// TwinCAT 3 PLC project TwinCAT_OpenFramework_Core
// Title: TwinCAT Open Framework Core
// Company: Oleksandr Tiutyk FOP
// Author: Oleksandr Tiutyk
// ProjectVersion: 0.0.0.1
// Description: Core types and implementations for TwinCAT Open Framework: abstractions, enums, primitives, interfaces, base object, exceptions, collettions, etc.
// ProgramVersion: 3.1.4026.16
// libraries:
//   Tc2_Standard, * (Beckhoff Automation GmbH)
//   Tc2_System, * (Beckhoff Automation GmbH)
//   Tc2_Utilities, * (Beckhoff Automation GmbH)
//   Tc3_EventLogger, * (Beckhoff Automation GmbH)
//   Tc3_JsonXml, * (Beckhoff Automation GmbH)
//   Tc3_Module, * (Beckhoff Automation GmbH)
// project tree:
//   Abstractions/Interfaces/Action/ IAbortableAction.TcIO, IAction.TcIO
//   Abstractions/Interfaces/ ICloneable.TcIO, IDisposable.TcIO, IObject.TcIO
//   Abstractions/Interfaces/Process/ IAbortableProcess.TcIO, IProcess.TcIO
//   Abstractions/ Object.TcPOU
//   Collections/PointerBased/PointerDictionary/ IReadOnlyPointerDictionary.TcIO, PointerDictionary.TcPOU, PointerDictionaryEnumerator.TcPOU
//   Collections/ Enumerator.TcPOU, ICollection.TcIO, IEnumerable.TcIO, IEnumerator.TcIO, KEY_VALUE_POINTER_PAIR.TcDUT
//   Collections/PointerBased/PointerUniqueSet/ IReadOnlyPointerUniqueSet.TcIO, PointerUniqueSet.TcPOU, PointerUniqueSetEnumerator.TcPOU
//   Collections/PointerBased/PointerList/ IReadOnlyPointerList.TcIO, PointerList.TcPOU, PointerListEnumerator.TcPOU
//   Collections/ValueBased/ByteList/ ByteList.TcPOU, ByteListEnumerator.TcPOU, IByteList.TcIO, IReadOnlyByteList.TcIO
//   Comparing/ COMPARISION_RESULT.TcDUT, IComparable.TcIO, IComparer.TcIO, StandardComparers.TcPOU
//   Comparing/StandardComparers/ BoolComparer.TcPOU, ByteComparer.TcPOU, DateAndTimeComparer.TcPOU, UXIntComparer.TcPOU, XIntComparer.TcPOU, XWordComparer.TcPOU, LDateAndTimeComparer.TcPOU, DateComparer.TcPOU, DIntComparer.TcPOU, DWordComparer.TcPOU, IntComparer.TcPOU, LIntComparer.TcPOU, LRealComparer.TcPOU, LTimeComparer.TcPOU, LWordComparer.TcPOU, PointerComparer.TcPOU, RealComparer.TcPOU, SIntComparer.TcPOU, StringComparer.TcPOU, TimeComparer.TcPOU, TimeOfDayComparer.TcPOU, LTimeOfDayComparer.TcPOU, UDIntComparer.TcPOU, UIntComparer.TcPOU, ULIntComparer.TcPOU, USIntComparer.TcPOU, WordComparer.TcPOU, WStringComparer.TcPOU
//   Enums/ EXECUTION_STATE.TcDUT, LOAD_STATE.TcDUT, POINTER_TYPE.TcDUT, SORTING_DIRECTION.TcDUT, TASK_STATE.TcDUT
//   Exceptions/Aggregate/ AggregateException.TcPOU
//   Exceptions/Empty/ EmptyException.TcPOU
//   Exceptions/ Exception.TcPOU, ExceptionManager.TcPOU, IException.TcIO
//   Exceptions/General/ArgumentOutOfRange/ ArgumentOutOfRangeException.TcPOU
//   Exceptions/General/ GeneralException.TcPOU
//   Exceptions/General/NotImplemented/ NotImplementedException.TcPOU
//   Exceptions/General/Standard/ StandardException.TcPOU
//   Exceptions/System/ SystemException.TcPOU
//   Helpers/ MathHelper.TcPOU
//   / CurrentNamespace.TcGVL
//   Internals/Statistics/ ObjectStatistics.TcPOU, ObjectStatisticsSettings.TcGVL, OBJECT_STATISTICS.TcDUT
//   Primitives/AnyType/ AnyTypeHelper.TcPOU
//   Primitives/Bit/ BitHelper.TcPOU
//   Primitives/Byte/ ByteHelper.TcPOU
//   Primitives/DateAndTime/ SystemDateTimeManager.TcPOU
//   Primitives/Pointer/ PointerHelper.TcPOU
//   Primitives/String/ StringBuilder.TcPOU, StringHelper.TcPOU
//   Primitives/WideString/ WideStringBuilder.TcPOU, WideStringHelper.TcPOU
//   Timers/ Timer.TcPOU
//   TypeAliases/ ERROR_MESSAGE.TcDUT, JSON_DOCUMENT.TcDUT

// ---- Collections/KEY_VALUE_POINTER_PAIR.TcDUT
TYPE KEY_VALUE_POINTER_PAIR :
STRUCT
	Key : PVOID;
	Value : PVOID;
END_STRUCT
END_TYPE

// ---- Comparing/COMPARISION_RESULT.TcDUT
{attribute 'qualified_only'}
{attribute 'strict'}
{attribute 'to_string'}
TYPE COMPARISION_RESULT :
(
	LEFT_LESS_RIGHT := -1,
	EQUALS := 0,
	LEFT_GREATER_RIGHT := 1
) SINT;
END_TYPE

// ---- Enums/EXECUTION_STATE.TcDUT
{attribute 'qualified_only'}
{attribute 'strict'}
{attribute 'to_string'}
// error should be reported using exceptions
TYPE EXECUTION_STATE :
(
	BUSY,
	DONE
);
END_TYPE

// ---- Enums/LOAD_STATE.TcDUT
{attribute 'qualified_only'}
{attribute 'strict'}
{attribute 'to_string'}
TYPE LOAD_STATE :
(
	NOT_LOADED,
	LOADING,
	LOADED,
	FAILED
);
END_TYPE

// ---- Enums/POINTER_TYPE.TcDUT
{attribute 'qualified_only'}
{attribute 'strict'}
{attribute 'to_string'}
TYPE POINTER_TYPE :
(
	BOOL_POINTER := 1,
	BYTE_POINTER := 2,
	WORD_POINTER := 3,
	DWORD_POINTER := 4,
	LWORD_POINTER := 5,
	SINT_POINTER := 6,
	USINT_POINTER := 7,
	INT_POINTER := 8,
	UINT_POINTER := 9,
	DINT_POINTER := 10,
	UDINT_POINTER := 11,
	LINT_POINTER := 12,
	ULINT_POINTER := 13,	
	XINT_POINTER := 14, 
	XWORD_POINTER := 15,	
	UXINT_POINTER := 16, 
	REAL_POINTER := 17,
	LREAL_POINTER := 18,
	STRING_POINTER := 19,
	WSTRING_POINTER := 20,
	TIME_POINTER := 21,
	LTIME_POINTER := 22,
	DATE_POINTER := 23,
	DATE_AND_TIME_POINTER := 24,
	LDATE_AND_TIME_POINTER := 25,
	TIME_OF_DAY_POINTER := 26,
	LTIME_OF_DAY_POINTER := 27,
	UNTYPED_POINTER := 28,
	OBJECT_POINTER := 29
) BYTE;
END_TYPE

// ---- Enums/SORTING_DIRECTION.TcDUT
{attribute 'qualified_only'}
{attribute 'strict'}
{attribute 'to_string'}
TYPE SORTING_DIRECTION :
(
	ASCENDING,
	DESCENDING
);
END_TYPE

// ---- Enums/TASK_STATE.TcDUT
{attribute 'qualified_only'}
{attribute 'strict'}
{attribute 'to_string'}
TYPE TASK_STATE :
(
	IDLE,
	EXECUTING,	
	DONE,
	ERROR,
	ABORTING,
	ABORTED
);
END_TYPE

// ---- Internals/Statistics/OBJECT_STATISTICS.TcDUT
TYPE OBJECT_STATISTICS :
STRUCT
	TypeName : STRING(255);
	InstanceCount : LINT;
END_STRUCT
END_TYPE

// ---- TypeAliases/ERROR_MESSAGE.TcDUT
TYPE ERROR_MESSAGE : WSTRING(2000); END_TYPE

// ---- TypeAliases/JSON_DOCUMENT.TcDUT
TYPE JSON_DOCUMENT : STRING(25000); END_TYPE

// ---- CurrentNamespace.TcGVL
{attribute 'qualified_only'}
VAR_GLOBAL
	{attribute 'OPC.UA.DA' := '1'}
	{attribute 'OPC.UA.DA.Access' := '1'}
	{attribute 'init_namespace'} 
	Name : STRING(255);	
END_VAR

// ---- Internals/Statistics/ObjectStatisticsSettings.TcGVL
{attribute 'qualified_only'}
VAR_GLOBAL PERSISTENT
	{attribute 'OPC.UA.DA' := '1'}	
	// Indicates if object creating and deleting counted in ObjectStatistics
	CountObjectStatistics : BOOL;
END_VAR

// ---- Abstractions/Interfaces/Action/IAbortableAction.TcIO
INTERFACE IAbortableAction EXTENDS IAction

{attribute 'monitoring' := 'call'}
{attribute 'OPC.UA.DA.Property' := '1'}
{attribute 'OPC.UA.DA.Access' := '1'}
PROPERTY Aborted : BOOL
GET
END_GET
END_PROPERTY

{attribute 'monitoring' := 'call'}
{attribute 'OPC.UA.DA.Property' := '1'}
{attribute 'OPC.UA.DA.Access' := '1'}
PROPERTY Aborting : BOOL
GET
END_GET
END_PROPERTY

{attribute 'monitoring' := 'call'}
{attribute 'OPC.UA.DA.Property' := '1'}
{attribute 'OPC.UA.DA.Access' := '1'}
PROPERTY AbortReason : REFERENCE TO ERROR_MESSAGE
GET
END_GET
END_PROPERTY

METHOD RequestAbort
VAR_INPUT 
	reason : ERROR_MESSAGE;
END_VAR
END_METHOD

END_INTERFACE

// ---- Abstractions/Interfaces/Action/IAction.TcIO
INTERFACE IAction EXTENDS IObject

{attribute 'monitoring' := 'call'}
{attribute 'OPC.UA.DA.Property' := '1'}
{attribute 'OPC.UA.DA.Access' := '1'}
PROPERTY Busy : BOOL
GET
END_GET
END_PROPERTY

{attribute 'monitoring' := 'call'}
{attribute 'OPC.UA.DA.Property' := '1'}
{attribute 'OPC.UA.DA.Access' := '1'}
PROPERTY Done : BOOL
GET
END_GET
END_PROPERTY

{attribute 'monitoring' := 'call'}
{attribute 'OPC.UA.DA.Property' := '1'}
{attribute 'OPC.UA.DA.Access' := '1'}
PROPERTY Error : BOOL
GET
END_GET
END_PROPERTY

METHOD Execute
END_METHOD

END_INTERFACE

// ---- Abstractions/Interfaces/ICloneable.TcIO
INTERFACE ICloneable EXTENDS __System.IQueryInterface

METHOD Clone : IObject
END_METHOD

END_INTERFACE

// ---- Abstractions/Interfaces/IDisposable.TcIO
INTERFACE IDisposable EXTENDS __System.IQueryInterface

METHOD Dispose
END_METHOD

END_INTERFACE

// ---- Abstractions/Interfaces/IObject.TcIO
INTERFACE IObject EXTENDS __System.IQueryInterface, IDisposable

{attribute 'monitoring' := 'call'}
PROPERTY ClassName : STRING
GET
END_GET
END_PROPERTY

{attribute "object_name" := "Equals"}
METHOD Equals : BOOL
VAR_INPUT 
	object : IObject;
END_VAR
END_METHOD

END_INTERFACE

// ---- Abstractions/Interfaces/Process/IAbortableProcess.TcIO
INTERFACE IAbortableProcess EXTENDS IProcess

{attribute 'monitoring' := 'call'}
{attribute 'OPC.UA.DA.Property' := '1'}
{attribute 'OPC.UA.DA.Access' := '1'}
PROPERTY Aborted : BOOL
GET
END_GET
END_PROPERTY

{attribute 'monitoring' := 'call'}
{attribute 'OPC.UA.DA.Property' := '1'}
{attribute 'OPC.UA.DA.Access' := '1'}
PROPERTY AbortReason : REFERENCE TO ERROR_MESSAGE
GET
END_GET
END_PROPERTY

{attribute 'monitoring' := 'call'}
{attribute 'OPC.UA.DA.Property' := '1'}
{attribute 'OPC.UA.DA.Access' := '1'}
PROPERTY Busy : BOOL
GET
END_GET
END_PROPERTY

METHOD RequestAbort
VAR_INPUT 
	reason : ERROR_MESSAGE;
END_VAR
END_METHOD

END_INTERFACE

// ---- Abstractions/Interfaces/Process/IProcess.TcIO
INTERFACE IProcess EXTENDS IObject

{attribute 'monitoring' := 'call'}
{attribute 'OPC.UA.DA.Property' := '1'}
{attribute 'OPC.UA.DA.Access' := '1'}
PROPERTY Busy : BOOL
GET
END_GET
END_PROPERTY

{attribute 'monitoring' := 'call'}
{attribute 'OPC.UA.DA.Property' := '1'}
{attribute 'OPC.UA.DA.Access' := '1'}
PROPERTY Error : BOOL
GET
END_GET
END_PROPERTY

METHOD Execute
END_METHOD

END_INTERFACE

// ---- Collections/PointerBased/PointerDictionary/IReadOnlyPointerDictionary.TcIO
INTERFACE IReadOnlyPointerDictionary EXTENDS ICollection

METHOD ContainsKey : BOOL
VAR_INPUT
	key : PVOID;
END_VAR
END_METHOD

METHOD GetKeyByIndex : PVOID
VAR_INPUT
	index : DINT;
END_VAR
END_METHOD

METHOD GetValueByIndex : PVOID
VAR_INPUT
	index : DINT;
END_VAR
END_METHOD

METHOD GetValueByKey : PVOID
VAR_INPUT
	key : PVOID;
END_VAR
END_METHOD

{attribute 'OPC.UA.DA.Property' := '1'}
{attribute 'monitoring' := 'call'}
PROPERTY KeyType : POINTER_TYPE
GET
END_GET
END_PROPERTY

{attribute 'OPC.UA.DA.Property' := '1'}
{attribute 'monitoring' := 'call'}
PROPERTY ValueType : POINTER_TYPE
GET
END_GET
END_PROPERTY

END_INTERFACE

// ---- Collections/PointerBased/PointerUniqueSet/IReadOnlyPointerUniqueSet.TcIO
INTERFACE IReadOnlyPointerUniqueSet EXTENDS ICollection

METHOD Contains : BOOL
VAR_INPUT
	element : PVOID;
END_VAR
END_METHOD

{attribute 'OPC.UA.DA.Property' := '1'}
{attribute 'monitoring' := 'call'}
PROPERTY ElementType : POINTER_TYPE
GET
END_GET
END_PROPERTY

METHOD GetByIndex : PVOID
VAR_INPUT
	index : DINT;
END_VAR
END_METHOD

END_INTERFACE

// ---- Collections/ICollection.TcIO
INTERFACE ICollection EXTENDS IEnumerable

{attribute 'OPC.UA.DA.Property' := '1'}
{attribute 'monitoring' := 'call'}
PROPERTY Count : DINT
GET
END_GET
END_PROPERTY

END_INTERFACE

// ---- Collections/IEnumerable.TcIO
INTERFACE IEnumerable EXTENDS IObject

METHOD GetDefaultEnumerator : IEnumerator
END_METHOD

END_INTERFACE

// ---- Collections/IEnumerator.TcIO
INTERFACE IEnumerator EXTENDS IObject

// Shows curent collection element
PROPERTY ABSTRACT Current : PVOID
GET
END_GET
END_PROPERTY

// Moves Current pointer to next collection element
METHOD MoveNext : BOOL
END_METHOD

// Sets the enumerator to its initial position, which is before the first element in the collection
METHOD Reset
END_METHOD

END_INTERFACE

// ---- Collections/PointerBased/PointerList/IReadOnlyPointerList.TcIO
INTERFACE IReadOnlyPointerList EXTENDS ICollection

{attribute 'OPC.UA.DA.Property' := '1'}
{attribute 'monitoring' := 'call'}
PROPERTY ElementType : POINTER_TYPE
GET
END_GET
END_PROPERTY

METHOD Find : BOOL
VAR_INPUT
	pattern : PVOID;
	comparer : IComparer;
	skip : DINT;
END_VAR
VAR_OUTPUT
	element : PVOID;
	index : DINT;
END_VAR
END_METHOD

METHOD Get : PVOID
VAR_INPUT
	index : DINT;
END_VAR
END_METHOD

METHOD Sort
VAR_INPUT
	comparer : IComparer;
	direction : SORTING_DIRECTION;
END_VAR
END_METHOD

END_INTERFACE

// ---- Collections/ValueBased/ByteList/IByteList.TcIO
INTERFACE IByteList EXTENDS IReadOnlyByteList

METHOD Set
VAR_INPUT
	index : DINT;
	value : BYTE;
END_VAR
END_METHOD

END_INTERFACE

// ---- Collections/ValueBased/ByteList/IReadOnlyByteList.TcIO
INTERFACE IReadOnlyByteList EXTENDS ICollection

{attribute 'OPC.UA.DA.Property' := '1'}
{attribute 'monitoring' := 'call'}
PROPERTY Address : POINTER TO BYTE
GET
END_GET
END_PROPERTY

METHOD Get : BYTE
VAR_INPUT
	index : DINT;
END_VAR
END_METHOD

END_INTERFACE

// ---- Comparing/IComparable.TcIO
INTERFACE IComparable EXTENDS IObject

METHOD CompareTo : COMPARISION_RESULT
VAR_INPUT
	object : IObject;
END_VAR
END_METHOD

END_INTERFACE

// ---- Comparing/IComparer.TcIO
INTERFACE IComparer EXTENDS IObject

METHOD Compare : COMPARISION_RESULT
VAR_INPUT
	left : PVOID;
	right : PVOID;
END_VAR
END_METHOD

END_INTERFACE

// ---- Exceptions/IException.TcIO
INTERFACE IException EXTENDS ICloneable, IDisposable

{attribute 'monitoring' := 'call'}
PROPERTY Empty : BOOL
GET
END_GET
END_PROPERTY

// Work is not possible after such error
{attribute 'monitoring' := 'call'}
PROPERTY Fatal : BOOL
GET
END_GET
END_PROPERTY

METHOD ABSTRACT GetMessage : ERROR_MESSAGE
VAR_INPUT
	showTimestamp : BOOL := FALSE;
	showSource : BOOL := FALSE;
END_VAR
END_METHOD

METHOD GetSourceDescription : WSTRING(300)
END_METHOD

{attribute 'monitoring' := 'call'}
PROPERTY LocalTimestamp : DATE_AND_TIME
GET
END_GET
END_PROPERTY

{attribute 'monitoring' := 'call'}
PROPERTY SourceClassName : STRING
GET
END_GET
END_PROPERTY

{attribute 'monitoring' := 'call'}
PROPERTY SourceMethodName : STRING
GET
END_GET
END_PROPERTY

{attribute 'monitoring' := 'call'}
PROPERTY SourceNamespaceName : STRING
GET
END_GET
END_PROPERTY

{attribute 'monitoring' := 'call'}
PROPERTY SourcePosition : STRING
GET
END_GET
END_PROPERTY

{attribute 'monitoring' := 'call'}
PROPERTY UtcTimestamp : DATE_AND_TIME
GET
END_GET
END_PROPERTY

END_INTERFACE

// ---- Abstractions/Object.TcPOU
{attribute 'no_explicit_call' := 'Direct call is not allowed'} 
FUNCTION_BLOCK ABSTRACT Object IMPLEMENTS IObject

{attribute 'monitoring' := 'call'}
PROPERTY ABSTRACT ClassName : STRING
GET
END_GET
END_PROPERTY

METHOD Dispose
VAR
	self : POINTER TO Object;
END_VAR
PointerHelper.ReleaseDynamicMemory(THIS, POINTER_TYPE.OBJECT_POINTER);
END_METHOD

{attribute "object_name" := "Equals"}
METHOD Equals : BOOL
VAR_INPUT 
	object : IObject;
END_VAR
VAR
	selfPointer : POINTER TO Object;
	comparingPointer : POINTER TO Object;
END_VAR
selfPointer := THIS;

IF __QUERYPOINTER(object, comparingPointer) THEN
	Equals := selfPointer = comparingPointer;
END_IF
END_METHOD

METHOD FB_exit : BOOL
VAR_INPUT
	bInCopyCode : BOOL; // if TRUE, the exit method is called for exiting an instance that is copied afterwards (online change).
END_VAR
IF ObjectStatisticsSettings.CountObjectStatistics THEN
	ObjectStatistics.RemoveObject(THIS^);
END_IF
END_METHOD

METHOD FB_init : BOOL
VAR_INPUT
	bInitRetains : BOOL; // if TRUE, the retain variables are initialized (warm start / cold start)
	bInCopyCode : BOOL; // if TRUE, the instance afterwards gets moved into the copy code (online change)
END_VAR
IF ObjectStatisticsSettings.CountObjectStatistics THEN
	ObjectStatistics.AddObject(THIS^);
END_IF
END_METHOD

END_FUNCTION_BLOCK

// ---- Primitives/Pointer/PointerHelper.TcPOU
PROGRAM PointerHelper

METHOD ReleaseDynamicMemory
VAR_INPUT
	value : POINTER TO BYTE;
	pointerType : POINTER_TYPE;
END_VAR
VAR
	memoryArea : Tc2_System.E_TcMemoryArea;
	objectPointer : POINTER TO Object;
END_VAR
IF value = 0 THEN
	RETURN;
END_IF

// check at list first byte of released memory
memoryArea := Tc2_System.F_CheckMemoryArea(value, 1);

IF memoryArea <> E_TcMemoryArea.Dynamic THEN
	RETURN;
END_IF

IF pointerType = POINTER_TYPE.OBJECT_POINTER THEN
	objectPointer := value;
	// to call FB_exit
	__DELETE(objectPointer);
ELSE
	__DELETE(value);
END_IF
END_METHOD

END_PROGRAM

// ---- Internals/Statistics/ObjectStatistics.TcPOU
{attribute 'no_explicit_call' := 'Direct call is not allowed'} 
PROGRAM ObjectStatistics
VAR CONSTANT
	{attribute 'OPC.UA.DA' := '1'}
	{attribute 'OPC.UA.DA.Access' := '1'}	
	OBJECT_STATISTICS_BUFFER_SIZE : DINT := 1000;
END_VAR
VAR_OUTPUT
	{attribute 'OPC.UA.DA' := '1'}
	{attribute 'OPC.UA.DA.Access' := '1'}	
	CreateObjectCounter : DWORD; // Increments each time when object created
	{attribute 'OPC.UA.DA' := '1'}
	{attribute 'OPC.UA.DA.Access' := '1'}	
	DeleteObjectCounter : DWORD; // Decrements each time when object created
	{attribute 'OPC.UA.DA' := '1'}
	{attribute 'OPC.UA.DA.Access' := '1'}	
	ObjectCount : LINT; // Count of existing objecs
	{attribute 'OPC.UA.DA' := '1'}
	{attribute 'OPC.UA.DA.Access' := '1'}	
	ObjectStatistics : ARRAY [0..OBJECT_STATISTICS_BUFFER_SIZE - 1] OF OBJECT_STATISTICS;
END_VAR

METHOD INTERNAL AddObject : BOOL
VAR_IN_OUT CONSTANT
	object : Object;
END_VAR
VAR
	i : DINT;
END_VAR
IF CreateObjectCounter < 4294967295 THEN
	CreateObjectCounter := CreateObjectCounter + 1;
ELSE
	CreateObjectCounter := 0;
END_IF

ObjectCount := ObjectCount + 1;

IF object.ClassName = '' THEN
	RETURN;	
END_IF

FOR i := 0 TO OBJECT_STATISTICS_BUFFER_SIZE - 1 DO
	IF ObjectStatistics[i].TypeName = object.ClassName THEN		
		ObjectStatistics[i].InstanceCount := ObjectStatistics[i].InstanceCount + 1;		
		RETURN;
	ELSIF ObjectStatistics[i].TypeName = '' THEN	
		ObjectStatistics[i].TypeName := object.ClassName;
		ObjectStatistics[i].InstanceCount := 1;		
		RETURN;
	END_IF
END_FOR
END_METHOD

METHOD INTERNAL RemoveObject
VAR_IN_OUT CONSTANT
	object : Object;
END_VAR
VAR
	i : DINT;
END_VAR
IF DeleteObjectCounter < 4294967295 THEN
	DeleteObjectCounter := DeleteObjectCounter + 1;
ELSE
	DeleteObjectCounter := 0;
END_IF

ObjectCount := ObjectCount - 1;

IF object.ClassName = '' THEN
	RETURN;	
END_IF

FOR i := 0 TO OBJECT_STATISTICS_BUFFER_SIZE - 1 DO
	IF ObjectStatistics[i].TypeName = object.ClassName THEN				
		ObjectStatistics[i].InstanceCount := ObjectStatistics[i].InstanceCount - 1;
						
		RETURN;
	END_IF 
END_FOR
END_METHOD

END_PROGRAM

// ---- Collections/PointerBased/PointerDictionary/PointerDictionary.TcPOU
{attribute 'no_explicit_call' := 'do not call this function block directly'} 
// Dynamic dictionary of pointers to key and value
FUNCTION_BLOCK PointerDictionary EXTENDS Object IMPLEMENTS IReadOnlyPointerDictionary
VAR
	_ClassName : STRING := __POUNAME();
	_Keys : POINTER TO PVOID;
	_Values : POINTER TO PVOID;
	_ArrayLength : DINT;
	_ElementCount : DINT;
	_DefaultAllocationElemetsCount : BYTE := 10;
	_KeyType : POINTER_TYPE := POINTER_TYPE.BYTE_POINTER;
	_ValueType : POINTER_TYPE := POINTER_TYPE.BYTE_POINTER;
	_KeyComparer : IComparer;
	_DefaultEnumerator : PointerDictionaryEnumerator;
END_VAR

METHOD AllocateMemory
VAR_INPUT
	elementsCount : DINT;
END_VAR
VAR
	newKeys : POINTER TO PVOID;
	newValues : POINTER TO PVOID;
END_VAR
newKeys := __NEW(PVOID, TO_UDINT(_ArrayLength + elementsCount));
newValues := __NEW(PVOID, TO_UDINT(_ArrayLength + elementsCount));

IF _ElementCount > 0 THEN
	Tc2_System.MEMCPY(newKeys, _Keys, SIZEOF(POINTER TO BYTE) * TO_UDINT(_ElementCount)); 
	Tc2_System.MEMCPY(newValues, _Values, SIZEOF(POINTER TO BYTE) * TO_UDINT(_ElementCount));
END_IF

IF _Keys <> 0 THEN
	__DELETE(_Keys);
END_IF

IF _Values <> 0 THEN
	__DELETE(_Values);
END_IF
 
_Keys := newKeys;
_Values := newValues;
 
_ArrayLength := _ArrayLength + elementsCount;
END_METHOD

{attribute 'monitoring' := 'call'}
PROPERTY ClassName : STRING
GET
ClassName := _ClassName;
END_GET
END_PROPERTY

METHOD Clear
VAR_INPUT
	deleteKeys : BOOL;
	deleteValues : BOOL;
END_VAR
VAR
	i : DINT;
	value : PVOID;
END_VAR
IF deleteKeys AND_THEN _ElementCount > 0 THEN
	FOR i := 0 TO _ElementCount - 1 DO
		PointerHelper.ReleaseDynamicMemory(_Keys[i], _KeyType);						
	END_FOR	
END_IF

IF deleteValues AND_THEN _ElementCount > 0 THEN
	FOR i := 0 TO _ElementCount - 1 DO
		PointerHelper.ReleaseDynamicMemory(_Values[i], _ValueType);							
	END_FOR	
END_IF

IF _Keys <> 0 THEN
	__DELETE(_Keys);
END_IF

IF _Values <> 0 THEN
	__DELETE(_Values);
END_IF

_ElementCount := 0;
_ArrayLength := 0;
END_METHOD

METHOD ContainsKey : BOOL
VAR_INPUT
	key : PVOID;
END_VAR
VAR
	index : DINT; 
END_VAR
ContainsKey := SearchKeyPosition(key, supposedIndex => index);
END_METHOD

{attribute 'OPC.UA.DA.Property' := '1'}
{attribute 'monitoring' := 'call'}
PROPERTY Count : DINT
GET
Count := _ElementCount;
END_GET
END_PROPERTY

METHOD FB_exit : BOOL
VAR_INPUT
	bInCopyCode : BOOL; // if TRUE, the exit method is called for exiting an instance that is copied afterwards (online change).
END_VAR
Clear(FALSE, FALSE);
END_METHOD

METHOD FB_init : BOOL
VAR_INPUT
	bInitRetains : BOOL; // if TRUE, the retain variables are initialized (warm start / cold start)
	bInCopyCode : BOOL; // if TRUE, the instance afterwards gets moved into the copy code (online change)
	keyType : POINTER_TYPE;
	valueType : POINTER_TYPE;
	keyComparer : IComparer;
END_VAR
_DefaultEnumerator.Initialize(THIS^);

_KeyType := keyType;
_ValueType := valueType;

IF keyComparer = 0 THEN
	_KeyComparer := StandardComparers.GetForType(keyType);
ELSE
	_KeyComparer := keyComparer;
END_IF
END_METHOD

METHOD GetDefaultEnumerator : IEnumerator
GetDefaultEnumerator := _DefaultEnumerator;
END_METHOD

METHOD GetKeyByIndex : PVOID
VAR_INPUT
	index : DINT;
END_VAR
IF index >= 0 AND index < _ElementCount THEN
	GetKeyByIndex := _Keys[index];
END_IF
END_METHOD

METHOD GetValueByIndex : PVOID
VAR_INPUT
	index : DINT;
END_VAR
IF index >= 0 AND index < _ElementCount THEN
	GetValueByIndex := _Values[index];
END_IF
END_METHOD

METHOD GetValueByKey : PVOID
VAR_INPUT
	key : PVOID;
END_VAR
VAR
	index : DINT; 
END_VAR
IF SearchKeyPosition(key, supposedIndex => index) THEN
	GetValueByKey := _Values[index];
END_IF
END_METHOD

{attribute 'OPC.UA.DA.Property' := '1'}
{attribute 'monitoring' := 'call'}
PROPERTY KeyType : POINTER_TYPE
GET
KeyType := _KeyType;
END_GET
END_PROPERTY

METHOD Remove : BOOL
VAR_INPUT
	key : PVOID;
	deleteKey : BOOL;
	deleteValue : BOOL;
END_VAR
VAR
	index : DINT;
END_VAR
IF SearchKeyPosition(key, supposedIndex => index) THEN
	RemoveAt(index, deleteKey, deleteValue);
	Remove := TRUE;
END_IF
END_METHOD

METHOD RemoveAt : BOOL
VAR_INPUT
	index : DINT;
	deleteKey : BOOL;
	deleteValue : BOOL;
END_VAR
VAR
	i : DINT;
END_VAR
IF index < _ElementCount THEN
	IF deleteKey THEN
		PointerHelper.ReleaseDynamicMemory(_Keys[index], _KeyType);			
	END_IF
	
	IF deleteValue THEN
		PointerHelper.ReleaseDynamicMemory(_Values[index], _ValueType);			
	END_IF
	
	IF index + 2 <= _ElementCount THEN
		FOR	i := index TO _ElementCount - 2 DO
			_Keys[i] := _Keys[i + 1];
			_Values[i] := _Values[i + 1];
		END_FOR			
	END_IF
		
	_Keys[_ElementCount - 1] := 0;
	_Values[_ElementCount - 1] := 0;
	_ElementCount := _ElementCount - 1;
	
	RemoveAt := TRUE;
END_IF
END_METHOD

METHOD PROTECTED SearchKeyPosition : BOOL
VAR_INPUT
	key : PVOID;
END_VAR
VAR_OUTPUT
	supposedIndex : DINT; 
END_VAR
VAR
	lastIndex : DINT;
	minIndex : DINT;
	maxIndex : DINT;
END_VAR
IF _ElementCount = 0 THEN
	RETURN;
END_IF

lastIndex := _ElementCount - 1;
maxIndex := lastIndex;
supposedIndex := maxIndex / 2;

WHILE minIndex <= maxIndex DO
	CASE _KeyComparer.Compare(_Keys[supposedIndex], key) OF
		// assumed key equals to seached 
		COMPARISION_RESULT.EQUALS:
			SearchKeyPosition := TRUE;
			RETURN;

		// assumed key less than searched, move range to right
		COMPARISION_RESULT.LEFT_LESS_RIGHT:
			minIndex := supposedIndex + 1;
			
		// assumed key greater than searched, move range to left	
		COMPARISION_RESULT.LEFT_GREATER_RIGHT:
			maxIndex := supposedIndex - 1;
	END_CASE
	
	supposedIndex := minIndex + (maxIndex - minIndex) / 2;
END_WHILE
END_METHOD

METHOD Set : DINT
VAR_INPUT
	key : PVOID;
	value : PVOID;
	deleteReplacedKey : BOOL;
	deleteReplacedValue : BOOL;
END_VAR
VAR
	index, i : DINT;
END_VAR
// if equal key found then we need to replace it
IF SearchKeyPosition(key, supposedIndex => index) THEN	
	// old and new keys show to diffirent address, then we need to replace existing key 
	IF _Keys[index] <> key THEN
		IF deleteReplacedKey THEN
			PointerHelper.ReleaseDynamicMemory(_Keys[index], _KeyType);
		END_IF
		
		_Keys[index] := key;
	END_IF
	
	// old and new values show to diffirent address, then we need to replace existing value 
	IF _Values[index] <> value THEN
		IF deleteReplacedValue THEN
			PointerHelper.ReleaseDynamicMemory(_Values[index], _ValueType);
		END_IF
		
		_Values[index] := value;
	END_IF
// if equal key not found than we need to insert it
ELSE
	IF _ElementCount >= _ArrayLength THEN
		AllocateMemory(_DefaultAllocationElemetsCount);
	END_IF
	
	i := _ElementCount;	
	_ElementCount := _ElementCount + 1;
		
	WHILE i > index DO
		_Keys[i] := _Keys[i - 1];
		_Values[i] := _Values[i - 1];
		
		i := i - 1;
	END_WHILE
	
	_Keys[index] := key;
	_Values[index] := value;
END_IF

Set := index;
END_METHOD

{attribute 'OPC.UA.DA.Property' := '1'}
{attribute 'monitoring' := 'call'}
PROPERTY ValueType : POINTER_TYPE
GET
ValueType := _ValueType;
END_GET
END_PROPERTY

END_FUNCTION_BLOCK

// ---- Collections/PointerBased/PointerDictionary/PointerDictionaryEnumerator.TcPOU
{attribute 'no_explicit_call' := 'do not call this function block directly'} 
{attribute 'enable_dynamic_creation'}
FUNCTION_BLOCK PointerDictionaryEnumerator EXTENDS Enumerator
VAR
	_ClassName : STRING := __POUNAME();
	_Dictionary : IReadOnlyPointerDictionary;
	_Current : KEY_VALUE_POINTER_PAIR;
END_VAR

{attribute 'monitoring' := 'call'}
PROPERTY ClassName : STRING
GET
ClassName := _ClassName;
END_GET
END_PROPERTY

{attribute 'OPC.UA.DA.Property' := '1'}
{attribute 'monitoring' := 'call'}
PROPERTY Current : PVOID
GET
Current := ADR(_Current);
END_GET
END_PROPERTY

{attribute 'OPC.UA.DA.Property' := '1'}
{attribute 'monitoring' := 'call'}
PROPERTY CurrentKeyValuePair : POINTER TO KEY_VALUE_POINTER_PAIR
GET
CurrentKeyValuePair := ADR(_Current);
END_GET
END_PROPERTY

METHOD INTERNAL Initialize 
VAR_INPUT
	dictionary : IReadOnlyPointerDictionary;
END_VAR
_Dictionary := dictionary;
END_METHOD

{attribute "object_name" := "MoveNext"}
METHOD MoveNext : BOOL
_CurrentIndex := _CurrentIndex + 1;

IF _CurrentIndex >= _Dictionary.Count THEN
	_Current.Key := 0;
	_Current.Value := 0;

	_CurrentIndex := _Dictionary.Count;
ELSE
	_Current.Key := _Dictionary.GetKeyByIndex(_CurrentIndex);
	_Current.Value := _Dictionary.GetValueByIndex(_CurrentIndex);
	
	MoveNext := TRUE;
END_IF
END_METHOD

{attribute "object_name" := "Reset"}
METHOD Reset
SUPER^.Reset();

_Current.Key := 0;
_Current.Value := 0;
END_METHOD

END_FUNCTION_BLOCK

// ---- Collections/Enumerator.TcPOU
{attribute 'no_explicit_call' := 'do not call this function block directly'} 
FUNCTION_BLOCK ABSTRACT Enumerator EXTENDS Object IMPLEMENTS IEnumerator
VAR
	_CurrentIndex : DINT := -1;
END_VAR

// Shows curent collection element
PROPERTY ABSTRACT Current : PVOID
GET
END_GET
END_PROPERTY

{attribute "object_name" := "MoveNext"}
// Moves Current pointer to next collection element
METHOD ABSTRACT MoveNext : BOOL
END_METHOD

{attribute "object_name" := "Reset"}
// Sets the enumerator to its initial position, which is before the first element in the collection
METHOD Reset
_CurrentIndex := -1;
END_METHOD

END_FUNCTION_BLOCK

// ---- Comparing/StandardComparers.TcPOU
PROGRAM StandardComparers
VAR
	_BoolComparer : BoolComparer;
	_ByteComparer : ByteComparer;
	_WordComparer : WordComparer;
	_DWordComparer : DWordComparer;
	_LWordComparer : LWordComparer;
	_SIntComparer : SIntComparer;
	_USIntComparer : USIntComparer;
	_IntComparer : IntComparer;
	_UIntComparer : UIntComparer;
	_DIntComparer : DIntComparer;
	_UDIntComparer : UDIntComparer;
	_LIntComparer : LIntComparer;
	_ULIntComparer : ULIntComparer;
	_UXIntComparer : UXIntComparer;
	_XIntComparer : XIntComparer;
	_XWordComparer : XWordComparer;	
	_RealComparer : RealComparer;
	_LRealComparer : LRealComparer;		
	_StringComparer : StringComparer;
	_WStringComparer : WStringComparer;
	_TimeComparer : TimeComparer;
	_LTimeComparer : LTimeComparer;
	_DateComparer : DateComparer;
	_DateAndTimeComparer : DateAndTimeComparer;
	_LDateAndTimeComparer : DateAndTimeComparer;
	_TimeOfDayComparer : TimeOfDayComparer;	
	_LTimeOfDayComparer : LTimeOfDayComparer;	
	_PointerComparer : PointerComparer;
END_VAR

METHOD GetForType : IComparer
VAR_INPUT
	pointerType : POINTER_TYPE;
END_VAR
VAR
	exception : ArgumentOutOfRangeException();
END_VAR
CASE pointerType OF
	POINTER_TYPE.BOOL_POINTER:
		GetForType := _BoolComparer;
	POINTER_TYPE.BYTE_POINTER:
		GetForType := _ByteComparer;
	POINTER_TYPE.WORD_POINTER:
		GetForType := _WordComparer;
	POINTER_TYPE.DWORD_POINTER:
		GetForType := _DWordComparer;
	POINTER_TYPE.LWORD_POINTER:
		GetForType := _LWordComparer;
	POINTER_TYPE.SINT_POINTER:
		GetForType := _SIntComparer;
	POINTER_TYPE.USINT_POINTER:
		GetForType := _USIntComparer;
	POINTER_TYPE.INT_POINTER:
		GetForType := _IntComparer;
	POINTER_TYPE.UINT_POINTER:
		GetForType := _UIntComparer;
	POINTER_TYPE.DINT_POINTER:
		GetForType := _DIntComparer;
	POINTER_TYPE.UDINT_POINTER:
		GetForType := _UDIntComparer;
	POINTER_TYPE.LINT_POINTER:
		GetForType := _LIntComparer;
	POINTER_TYPE.ULINT_POINTER:
		GetForType := _ULIntComparer;
	POINTER_TYPE.XINT_POINTER:
		GetForType := _XIntComparer;
	POINTER_TYPE.XWORD_POINTER:
		GetForType := _XWordComparer;
	POINTER_TYPE.UXINT_POINTER:
		GetForType := _UXIntComparer;		
	POINTER_TYPE.REAL_POINTER:
		GetForType := _RealComparer;
	POINTER_TYPE.LREAL_POINTER:
		GetForType := _LRealComparer;
	POINTER_TYPE.STRING_POINTER:
		GetForType := _StringComparer;
	POINTER_TYPE.WSTRING_POINTER:
		GetForType := _WStringComparer;
	POINTER_TYPE.TIME_POINTER:
		GetForType := _TimeComparer;
	POINTER_TYPE.LTIME_POINTER:
		GetForType := _LTimeComparer;
	POINTER_TYPE.DATE_POINTER:
		GetForType := _DateComparer;
	POINTER_TYPE.DATE_AND_TIME_POINTER:
		GetForType := _DateAndTimeComparer;
	POINTER_TYPE.LDATE_AND_TIME_POINTER:
		GetForType := _LDateAndTimeComparer;
	POINTER_TYPE.TIME_OF_DAY_POINTER:
		GetForType := _TimeOfDayComparer;
	POINTER_TYPE.LTIME_OF_DAY_POINTER:
		GetForType := _LTimeOfDayComparer;
	POINTER_TYPE.UNTYPED_POINTER:
		GetForType := _PointerComparer;
	POINTER_TYPE.OBJECT_POINTER:
		GetForType := _PointerComparer;
	ELSE
		exception.Throw(CurrentNamespace.Name, 'StandardComparers', __POUNAME(), __POSITION(), 'pointerType', pointerType);
END_CASE
END_METHOD

END_PROGRAM

// ---- Comparing/StandardComparers/BoolComparer.TcPOU
FUNCTION_BLOCK BoolComparer EXTENDS Object IMPLEMENTS IComparer
VAR
	_ClassName : STRING := __POUNAME();
END_VAR

{attribute 'monitoring' := 'call'}
PROPERTY ClassName : STRING
GET
ClassName := _ClassName;
END_GET
END_PROPERTY

{attribute "object_name" := "Compare"}
METHOD Compare : COMPARISION_RESULT
VAR_INPUT
	left : PVOID;
	right : PVOID;
END_VAR
VAR
	leftPointer : POINTER TO BOOL; 
	rightPointer : POINTER TO BOOL; 
END_VAR
IF left = 0 AND right = 0 THEN
	Compare := COMPARISION_RESULT.EQUALS;
	RETURN;
END_IF

IF left = 0 THEN
	Compare := COMPARISION_RESULT.LEFT_LESS_RIGHT;
	RETURN;	
END_IF

IF right = 0 THEN
	Compare := COMPARISION_RESULT.LEFT_GREATER_RIGHT;
	RETURN;	
END_IF

leftPointer := left;
rightPointer := right;

IF leftPointer^ < rightPointer^ THEN
	Compare := COMPARISION_RESULT.LEFT_LESS_RIGHT;
ELSIF leftPointer^ > rightPointer^ THEN
	Compare := COMPARISION_RESULT.LEFT_GREATER_RIGHT;
ELSE
	Compare := COMPARISION_RESULT.EQUALS;	
END_IF
END_METHOD

END_FUNCTION_BLOCK

// ---- Comparing/StandardComparers/ByteComparer.TcPOU
FUNCTION_BLOCK ByteComparer EXTENDS Object IMPLEMENTS IComparer
VAR
	_ClassName : STRING := __POUNAME();
END_VAR

{attribute 'monitoring' := 'call'}
PROPERTY ClassName : STRING
GET
ClassName := _ClassName;
END_GET
END_PROPERTY

{attribute "object_name" := "Compare"}
METHOD Compare : COMPARISION_RESULT
VAR_INPUT
	left : PVOID;
	right : PVOID;
END_VAR
VAR
	leftPointer : POINTER TO BYTE; 
	rightPointer : POINTER TO BYTE; 
END_VAR
IF left = 0 AND right = 0 THEN
	Compare := COMPARISION_RESULT.EQUALS;
	RETURN;
END_IF

IF left = 0 THEN
	Compare := COMPARISION_RESULT.LEFT_LESS_RIGHT;
	RETURN;	
END_IF

IF right = 0 THEN
	Compare := COMPARISION_RESULT.LEFT_GREATER_RIGHT;
	RETURN;	
END_IF

leftPointer := left;
rightPointer := right;

IF leftPointer^ < rightPointer^ THEN
	Compare := COMPARISION_RESULT.LEFT_LESS_RIGHT;
ELSIF leftPointer^ > rightPointer^ THEN
	Compare := COMPARISION_RESULT.LEFT_GREATER_RIGHT;
ELSE
	Compare := COMPARISION_RESULT.EQUALS;	
END_IF
END_METHOD

END_FUNCTION_BLOCK

// ---- Comparing/StandardComparers/WordComparer.TcPOU
FUNCTION_BLOCK WordComparer EXTENDS Object IMPLEMENTS IComparer
VAR
	_ClassName : STRING := __POUNAME();
END_VAR

{attribute 'monitoring' := 'call'}
PROPERTY ClassName : STRING
GET
ClassName := _ClassName;
END_GET
END_PROPERTY

{attribute "object_name" := "Compare"}
METHOD Compare : COMPARISION_RESULT
VAR_INPUT
	left : PVOID;
	right : PVOID;
END_VAR
VAR
	leftPointer : POINTER TO WORD; 
	rightPointer : POINTER TO WORD; 
END_VAR
IF left = 0 AND right = 0 THEN
	Compare := COMPARISION_RESULT.EQUALS;
	RETURN;
END_IF

IF left = 0 THEN
	Compare := COMPARISION_RESULT.LEFT_LESS_RIGHT;
	RETURN;	
END_IF

IF right = 0 THEN
	Compare := COMPARISION_RESULT.LEFT_GREATER_RIGHT;
	RETURN;	
END_IF

leftPointer := left;
rightPointer := right;

IF leftPointer^ < rightPointer^ THEN
	Compare := COMPARISION_RESULT.LEFT_LESS_RIGHT;
ELSIF leftPointer^ > rightPointer^ THEN
	Compare := COMPARISION_RESULT.LEFT_GREATER_RIGHT;
ELSE
	Compare := COMPARISION_RESULT.EQUALS;	
END_IF
END_METHOD

END_FUNCTION_BLOCK

// ---- Comparing/StandardComparers/DWordComparer.TcPOU
FUNCTION_BLOCK DWordComparer EXTENDS Object IMPLEMENTS IComparer
VAR
	_ClassName : STRING := __POUNAME();
END_VAR

{attribute 'monitoring' := 'call'}
PROPERTY ClassName : STRING
GET
ClassName := _ClassName;
END_GET
END_PROPERTY

{attribute "object_name" := "Compare"}
METHOD Compare : COMPARISION_RESULT
VAR_INPUT
	left : PVOID;
	right : PVOID;
END_VAR
VAR
	leftPointer : POINTER TO DWORD; 
	rightPointer : POINTER TO DWORD; 
END_VAR
IF left = 0 AND right = 0 THEN
	Compare := COMPARISION_RESULT.EQUALS;
	RETURN;
END_IF

IF left = 0 THEN
	Compare := COMPARISION_RESULT.LEFT_LESS_RIGHT;
	RETURN;	
END_IF

IF right = 0 THEN
	Compare := COMPARISION_RESULT.LEFT_GREATER_RIGHT;
	RETURN;	
END_IF

leftPointer := left;
rightPointer := right;

IF leftPointer^ < rightPointer^ THEN
	Compare := COMPARISION_RESULT.LEFT_LESS_RIGHT;
ELSIF leftPointer^ > rightPointer^ THEN
	Compare := COMPARISION_RESULT.LEFT_GREATER_RIGHT;
ELSE
	Compare := COMPARISION_RESULT.EQUALS;	
END_IF
END_METHOD

END_FUNCTION_BLOCK

// ---- Comparing/StandardComparers/LWordComparer.TcPOU
FUNCTION_BLOCK LWordComparer EXTENDS Object IMPLEMENTS IComparer
VAR
	_ClassName : STRING := __POUNAME();
END_VAR

{attribute 'monitoring' := 'call'}
PROPERTY ClassName : STRING
GET
ClassName := _ClassName;
END_GET
END_PROPERTY

{attribute "object_name" := "Compare"}
METHOD Compare : COMPARISION_RESULT
VAR_INPUT
	left : PVOID;
	right : PVOID;
END_VAR
VAR
	leftPointer : POINTER TO LWORD; 
	rightPointer : POINTER TO LWORD; 
END_VAR
IF left = 0 AND right = 0 THEN
	Compare := COMPARISION_RESULT.EQUALS;
	RETURN;
END_IF

IF left = 0 THEN
	Compare := COMPARISION_RESULT.LEFT_LESS_RIGHT;
	RETURN;	
END_IF

IF right = 0 THEN
	Compare := COMPARISION_RESULT.LEFT_GREATER_RIGHT;
	RETURN;	
END_IF

leftPointer := left;
rightPointer := right;

IF leftPointer^ < rightPointer^ THEN
	Compare := COMPARISION_RESULT.LEFT_LESS_RIGHT;
ELSIF leftPointer^ > rightPointer^ THEN
	Compare := COMPARISION_RESULT.LEFT_GREATER_RIGHT;
ELSE
	Compare := COMPARISION_RESULT.EQUALS;	
END_IF
END_METHOD

END_FUNCTION_BLOCK

// ---- Comparing/StandardComparers/SIntComparer.TcPOU
FUNCTION_BLOCK SIntComparer EXTENDS Object IMPLEMENTS IComparer
VAR
	_ClassName : STRING := __POUNAME();
END_VAR

{attribute 'monitoring' := 'call'}
PROPERTY ClassName : STRING
GET
ClassName := _ClassName;
END_GET
END_PROPERTY

{attribute "object_name" := "Compare"}
METHOD Compare : COMPARISION_RESULT
VAR_INPUT
	left : PVOID;
	right : PVOID;
END_VAR
VAR
	leftPointer : POINTER TO SINT; 
	rightPointer : POINTER TO SINT; 
END_VAR
IF left = 0 AND right = 0 THEN
	Compare := COMPARISION_RESULT.EQUALS;
	RETURN;
END_IF

IF left = 0 THEN
	Compare := COMPARISION_RESULT.LEFT_LESS_RIGHT;
	RETURN;	
END_IF

IF right = 0 THEN
	Compare := COMPARISION_RESULT.LEFT_GREATER_RIGHT;
	RETURN;	
END_IF

leftPointer := left;
rightPointer := right;

IF leftPointer^ < rightPointer^ THEN
	Compare := COMPARISION_RESULT.LEFT_LESS_RIGHT;
ELSIF leftPointer^ > rightPointer^ THEN
	Compare := COMPARISION_RESULT.LEFT_GREATER_RIGHT;
ELSE
	Compare := COMPARISION_RESULT.EQUALS;	
END_IF
END_METHOD

END_FUNCTION_BLOCK

// ---- Comparing/StandardComparers/USIntComparer.TcPOU
FUNCTION_BLOCK USIntComparer EXTENDS Object IMPLEMENTS IComparer
VAR
	_ClassName : STRING := __POUNAME();
END_VAR

{attribute 'monitoring' := 'call'}
PROPERTY ClassName : STRING
GET
ClassName := _ClassName;
END_GET
END_PROPERTY

{attribute "object_name" := "Compare"}
METHOD Compare : COMPARISION_RESULT
VAR_INPUT
	left : PVOID;
	right : PVOID;
END_VAR
VAR
	leftPointer : POINTER TO USINT; 
	rightPointer : POINTER TO USINT; 
END_VAR
IF left = 0 AND right = 0 THEN
	Compare := COMPARISION_RESULT.EQUALS;
	RETURN;
END_IF

IF left = 0 THEN
	Compare := COMPARISION_RESULT.LEFT_LESS_RIGHT;
	RETURN;	
END_IF

IF right = 0 THEN
	Compare := COMPARISION_RESULT.LEFT_GREATER_RIGHT;
	RETURN;	
END_IF

leftPointer := left;
rightPointer := right;

IF leftPointer^ < rightPointer^ THEN
	Compare := COMPARISION_RESULT.LEFT_LESS_RIGHT;
ELSIF leftPointer^ > rightPointer^ THEN
	Compare := COMPARISION_RESULT.LEFT_GREATER_RIGHT;
ELSE
	Compare := COMPARISION_RESULT.EQUALS;	
END_IF
END_METHOD

END_FUNCTION_BLOCK

// ---- Comparing/StandardComparers/IntComparer.TcPOU
FUNCTION_BLOCK IntComparer EXTENDS Object IMPLEMENTS IComparer
VAR
	_ClassName : STRING := __POUNAME();
END_VAR

{attribute 'monitoring' := 'call'}
PROPERTY ClassName : STRING
GET
ClassName := _ClassName;
END_GET
END_PROPERTY

{attribute "object_name" := "Compare"}
METHOD Compare : COMPARISION_RESULT
VAR_INPUT
	left : PVOID;
	right : PVOID;
END_VAR
VAR
	leftPointer : POINTER TO INT; 
	rightPointer : POINTER TO INT; 
END_VAR
IF left = 0 AND right = 0 THEN
	Compare := COMPARISION_RESULT.EQUALS;
	RETURN;
END_IF

IF left = 0 THEN
	Compare := COMPARISION_RESULT.LEFT_LESS_RIGHT;
	RETURN;	
END_IF

IF right = 0 THEN
	Compare := COMPARISION_RESULT.LEFT_GREATER_RIGHT;
	RETURN;	
END_IF

leftPointer := left;
rightPointer := right;

IF leftPointer^ < rightPointer^ THEN
	Compare := COMPARISION_RESULT.LEFT_LESS_RIGHT;
ELSIF leftPointer^ > rightPointer^ THEN
	Compare := COMPARISION_RESULT.LEFT_GREATER_RIGHT;
ELSE
	Compare := COMPARISION_RESULT.EQUALS;	
END_IF
END_METHOD

END_FUNCTION_BLOCK

// ---- Comparing/StandardComparers/UIntComparer.TcPOU
FUNCTION_BLOCK UIntComparer EXTENDS Object IMPLEMENTS IComparer
VAR
	_ClassName : STRING := __POUNAME();
END_VAR

{attribute 'monitoring' := 'call'}
PROPERTY ClassName : STRING
GET
ClassName := _ClassName;
END_GET
END_PROPERTY

{attribute "object_name" := "Compare"}
METHOD Compare : COMPARISION_RESULT
VAR_INPUT
	left : PVOID;
	right : PVOID;
END_VAR
VAR
	leftPointer : POINTER TO UINT; 
	rightPointer : POINTER TO UINT; 
END_VAR
IF left = 0 AND right = 0 THEN
	Compare := COMPARISION_RESULT.EQUALS;
	RETURN;
END_IF

IF left = 0 THEN
	Compare := COMPARISION_RESULT.LEFT_LESS_RIGHT;
	RETURN;	
END_IF

IF right = 0 THEN
	Compare := COMPARISION_RESULT.LEFT_GREATER_RIGHT;
	RETURN;	
END_IF

leftPointer := left;
rightPointer := right;

IF leftPointer^ < rightPointer^ THEN
	Compare := COMPARISION_RESULT.LEFT_LESS_RIGHT;
ELSIF leftPointer^ > rightPointer^ THEN
	Compare := COMPARISION_RESULT.LEFT_GREATER_RIGHT;
ELSE
	Compare := COMPARISION_RESULT.EQUALS;	
END_IF
END_METHOD

END_FUNCTION_BLOCK

// ---- Comparing/StandardComparers/DIntComparer.TcPOU
FUNCTION_BLOCK DIntComparer EXTENDS Object IMPLEMENTS IComparer
VAR
	_ClassName : STRING := __POUNAME();
END_VAR

{attribute 'monitoring' := 'call'}
PROPERTY ClassName : STRING
GET
ClassName := _ClassName;
END_GET
END_PROPERTY

{attribute "object_name" := "Compare"}
METHOD Compare : COMPARISION_RESULT
VAR_INPUT
	left : PVOID;
	right : PVOID;
END_VAR
VAR
	leftPointer : POINTER TO DINT; 
	rightPointer : POINTER TO DINT; 
END_VAR
IF left = 0 AND right = 0 THEN
	Compare := COMPARISION_RESULT.EQUALS;
	RETURN;
END_IF

IF left = 0 THEN
	Compare := COMPARISION_RESULT.LEFT_LESS_RIGHT;
	RETURN;	
END_IF

IF right = 0 THEN
	Compare := COMPARISION_RESULT.LEFT_GREATER_RIGHT;
	RETURN;	
END_IF

leftPointer := left;
rightPointer := right;

IF leftPointer^ < rightPointer^ THEN
	Compare := COMPARISION_RESULT.LEFT_LESS_RIGHT;
ELSIF leftPointer^ > rightPointer^ THEN
	Compare := COMPARISION_RESULT.LEFT_GREATER_RIGHT;
ELSE
	Compare := COMPARISION_RESULT.EQUALS;	
END_IF
END_METHOD

END_FUNCTION_BLOCK

// ---- Comparing/StandardComparers/UDIntComparer.TcPOU
FUNCTION_BLOCK UDIntComparer EXTENDS Object IMPLEMENTS IComparer
VAR
	_ClassName : STRING := __POUNAME();
END_VAR

{attribute 'monitoring' := 'call'}
PROPERTY ClassName : STRING
GET
ClassName := _ClassName;
END_GET
END_PROPERTY

{attribute "object_name" := "Compare"}
METHOD Compare : COMPARISION_RESULT
VAR_INPUT
	left : PVOID;
	right : PVOID;
END_VAR
VAR
	leftPointer : POINTER TO UDINT; 
	rightPointer : POINTER TO UDINT; 
END_VAR
IF left = 0 AND right = 0 THEN
	Compare := COMPARISION_RESULT.EQUALS;
	RETURN;
END_IF

IF left = 0 THEN
	Compare := COMPARISION_RESULT.LEFT_LESS_RIGHT;
	RETURN;	
END_IF

IF right = 0 THEN
	Compare := COMPARISION_RESULT.LEFT_GREATER_RIGHT;
	RETURN;	
END_IF

leftPointer := left;
rightPointer := right;

IF leftPointer^ < rightPointer^ THEN
	Compare := COMPARISION_RESULT.LEFT_LESS_RIGHT;
ELSIF leftPointer^ > rightPointer^ THEN
	Compare := COMPARISION_RESULT.LEFT_GREATER_RIGHT;
ELSE
	Compare := COMPARISION_RESULT.EQUALS;	
END_IF
END_METHOD

END_FUNCTION_BLOCK

// ---- Comparing/StandardComparers/LIntComparer.TcPOU
FUNCTION_BLOCK LIntComparer EXTENDS Object IMPLEMENTS IComparer
VAR
	_ClassName : STRING := __POUNAME();
END_VAR

{attribute 'monitoring' := 'call'}
PROPERTY ClassName : STRING
GET
ClassName := _ClassName;
END_GET
END_PROPERTY

{attribute "object_name" := "Compare"}
METHOD Compare : COMPARISION_RESULT
VAR_INPUT
	left : PVOID;
	right : PVOID;
END_VAR
VAR
	leftPointer : POINTER TO LINT; 
	rightPointer : POINTER TO LINT; 
END_VAR
IF left = 0 AND right = 0 THEN
	Compare := COMPARISION_RESULT.EQUALS;
	RETURN;
END_IF

IF left = 0 THEN
	Compare := COMPARISION_RESULT.LEFT_LESS_RIGHT;
	RETURN;	
END_IF

IF right = 0 THEN
	Compare := COMPARISION_RESULT.LEFT_GREATER_RIGHT;
	RETURN;	
END_IF

leftPointer := left;
rightPointer := right;

IF leftPointer^ < rightPointer^ THEN
	Compare := COMPARISION_RESULT.LEFT_LESS_RIGHT;
ELSIF leftPointer^ > rightPointer^ THEN
	Compare := COMPARISION_RESULT.LEFT_GREATER_RIGHT;
ELSE
	Compare := COMPARISION_RESULT.EQUALS;	
END_IF
END_METHOD

END_FUNCTION_BLOCK

// ---- Comparing/StandardComparers/ULIntComparer.TcPOU
FUNCTION_BLOCK ULIntComparer EXTENDS Object IMPLEMENTS IComparer
VAR
	_ClassName : STRING := __POUNAME();
END_VAR

{attribute 'monitoring' := 'call'}
PROPERTY ClassName : STRING
GET
ClassName := _ClassName;
END_GET
END_PROPERTY

{attribute "object_name" := "Compare"}
METHOD Compare : COMPARISION_RESULT
VAR_INPUT
	left : PVOID;
	right : PVOID;
END_VAR
VAR
	leftPointer : POINTER TO ULINT; 
	rightPointer : POINTER TO ULINT; 
END_VAR
IF left = 0 AND right = 0 THEN
	Compare := COMPARISION_RESULT.EQUALS;
	RETURN;
END_IF

IF left = 0 THEN
	Compare := COMPARISION_RESULT.LEFT_LESS_RIGHT;
	RETURN;	
END_IF

IF right = 0 THEN
	Compare := COMPARISION_RESULT.LEFT_GREATER_RIGHT;
	RETURN;	
END_IF

leftPointer := left;
rightPointer := right;

IF leftPointer^ < rightPointer^ THEN
	Compare := COMPARISION_RESULT.LEFT_LESS_RIGHT;
ELSIF leftPointer^ > rightPointer^ THEN
	Compare := COMPARISION_RESULT.LEFT_GREATER_RIGHT;
ELSE
	Compare := COMPARISION_RESULT.EQUALS;	
END_IF
END_METHOD

END_FUNCTION_BLOCK

// ---- Comparing/StandardComparers/UXIntComparer.TcPOU
FUNCTION_BLOCK UXIntComparer EXTENDS Object IMPLEMENTS IComparer
VAR
	_ClassName : STRING := __POUNAME();
END_VAR

{attribute 'monitoring' := 'call'}
PROPERTY ClassName : STRING
GET
ClassName := _ClassName;
END_GET
END_PROPERTY

{attribute "object_name" := "Compare"}
METHOD Compare : COMPARISION_RESULT
VAR_INPUT
	left : PVOID;
	right : PVOID;
END_VAR
VAR
	leftPointer : POINTER TO __UXINT; 
	rightPointer : POINTER TO __UXINT; 
END_VAR
IF left = 0 AND right = 0 THEN
	Compare := COMPARISION_RESULT.EQUALS;
	RETURN;
END_IF

IF left = 0 THEN
	Compare := COMPARISION_RESULT.LEFT_LESS_RIGHT;
	RETURN;	
END_IF

IF right = 0 THEN
	Compare := COMPARISION_RESULT.LEFT_GREATER_RIGHT;
	RETURN;	
END_IF

leftPointer := left;
rightPointer := right;

IF leftPointer^ < rightPointer^ THEN
	Compare := COMPARISION_RESULT.LEFT_LESS_RIGHT;
ELSIF leftPointer^ > rightPointer^ THEN
	Compare := COMPARISION_RESULT.LEFT_GREATER_RIGHT;
ELSE
	Compare := COMPARISION_RESULT.EQUALS;	
END_IF
END_METHOD

END_FUNCTION_BLOCK

// ---- Comparing/StandardComparers/XIntComparer.TcPOU
FUNCTION_BLOCK XIntComparer EXTENDS Object IMPLEMENTS IComparer
VAR
	_ClassName : STRING := __POUNAME();
END_VAR

{attribute 'monitoring' := 'call'}
PROPERTY ClassName : STRING
GET
ClassName := _ClassName;
END_GET
END_PROPERTY

{attribute "object_name" := "Compare"}
METHOD Compare : COMPARISION_RESULT
VAR_INPUT
	left : PVOID;
	right : PVOID;
END_VAR
VAR
	leftPointer : POINTER TO __XINT; 
	rightPointer : POINTER TO __XINT; 
END_VAR
IF left = 0 AND right = 0 THEN
	Compare := COMPARISION_RESULT.EQUALS;
	RETURN;
END_IF

IF left = 0 THEN
	Compare := COMPARISION_RESULT.LEFT_LESS_RIGHT;
	RETURN;	
END_IF

IF right = 0 THEN
	Compare := COMPARISION_RESULT.LEFT_GREATER_RIGHT;
	RETURN;	
END_IF

leftPointer := left;
rightPointer := right;

IF leftPointer^ < rightPointer^ THEN
	Compare := COMPARISION_RESULT.LEFT_LESS_RIGHT;
ELSIF leftPointer^ > rightPointer^ THEN
	Compare := COMPARISION_RESULT.LEFT_GREATER_RIGHT;
ELSE
	Compare := COMPARISION_RESULT.EQUALS;	
END_IF
END_METHOD

END_FUNCTION_BLOCK

// ---- Comparing/StandardComparers/XWordComparer.TcPOU
FUNCTION_BLOCK XWordComparer EXTENDS Object IMPLEMENTS IComparer
VAR
	_ClassName : STRING := __POUNAME();
END_VAR

{attribute 'monitoring' := 'call'}
PROPERTY ClassName : STRING
GET
ClassName := _ClassName;
END_GET
END_PROPERTY

{attribute "object_name" := "Compare"}
METHOD Compare : COMPARISION_RESULT
VAR_INPUT
	left : PVOID;
	right : PVOID;
END_VAR
VAR
	leftPointer : POINTER TO __XWORD; 
	rightPointer : POINTER TO __XWORD; 
END_VAR
IF left = 0 AND right = 0 THEN
	Compare := COMPARISION_RESULT.EQUALS;
	RETURN;
END_IF

IF left = 0 THEN
	Compare := COMPARISION_RESULT.LEFT_LESS_RIGHT;
	RETURN;	
END_IF

IF right = 0 THEN
	Compare := COMPARISION_RESULT.LEFT_GREATER_RIGHT;
	RETURN;	
END_IF

leftPointer := left;
rightPointer := right;

IF leftPointer^ < rightPointer^ THEN
	Compare := COMPARISION_RESULT.LEFT_LESS_RIGHT;
ELSIF leftPointer^ > rightPointer^ THEN
	Compare := COMPARISION_RESULT.LEFT_GREATER_RIGHT;
ELSE
	Compare := COMPARISION_RESULT.EQUALS;	
END_IF
END_METHOD

END_FUNCTION_BLOCK

// ---- Comparing/StandardComparers/RealComparer.TcPOU
FUNCTION_BLOCK RealComparer EXTENDS Object IMPLEMENTS IComparer
VAR
	_ClassName : STRING := __POUNAME();
END_VAR

{attribute 'monitoring' := 'call'}
PROPERTY ClassName : STRING
GET
ClassName := _ClassName;
END_GET
END_PROPERTY

{attribute "object_name" := "Compare"}
METHOD Compare : COMPARISION_RESULT
VAR_INPUT
	left : PVOID;
	right : PVOID;
END_VAR
VAR
	leftPointer : POINTER TO REAL; 
	rightPointer : POINTER TO REAL; 
END_VAR
IF left = 0 AND right = 0 THEN
	Compare := COMPARISION_RESULT.EQUALS;
	RETURN;
END_IF

IF left = 0 THEN
	Compare := COMPARISION_RESULT.LEFT_LESS_RIGHT;
	RETURN;	
END_IF

IF right = 0 THEN
	Compare := COMPARISION_RESULT.LEFT_GREATER_RIGHT;
	RETURN;	
END_IF

leftPointer := left;
rightPointer := right;

IF leftPointer^ < rightPointer^ THEN
	Compare := COMPARISION_RESULT.LEFT_LESS_RIGHT;
ELSIF leftPointer^ > rightPointer^ THEN
	Compare := COMPARISION_RESULT.LEFT_GREATER_RIGHT;
ELSE
	Compare := COMPARISION_RESULT.EQUALS;	
END_IF
END_METHOD

END_FUNCTION_BLOCK

// ---- Comparing/StandardComparers/LRealComparer.TcPOU
FUNCTION_BLOCK LRealComparer EXTENDS Object IMPLEMENTS IComparer
VAR
	_ClassName : STRING := __POUNAME();
END_VAR

{attribute 'monitoring' := 'call'}
PROPERTY ClassName : STRING
GET
ClassName := _ClassName;
END_GET
END_PROPERTY

{attribute "object_name" := "Compare"}
METHOD Compare : COMPARISION_RESULT
VAR_INPUT
	left : PVOID;
	right : PVOID;
END_VAR
VAR
	leftPointer : POINTER TO LREAL; 
	rightPointer : POINTER TO LREAL; 
END_VAR
IF left = 0 AND right = 0 THEN
	Compare := COMPARISION_RESULT.EQUALS;
	RETURN;
END_IF

IF left = 0 THEN
	Compare := COMPARISION_RESULT.LEFT_LESS_RIGHT;
	RETURN;	
END_IF

IF right = 0 THEN
	Compare := COMPARISION_RESULT.LEFT_GREATER_RIGHT;
	RETURN;	
END_IF

leftPointer := left;
rightPointer := right;

IF leftPointer^ < rightPointer^ THEN
	Compare := COMPARISION_RESULT.LEFT_LESS_RIGHT;
ELSIF leftPointer^ > rightPointer^ THEN
	Compare := COMPARISION_RESULT.LEFT_GREATER_RIGHT;
ELSE
	Compare := COMPARISION_RESULT.EQUALS;	
END_IF
END_METHOD

END_FUNCTION_BLOCK

// ---- Comparing/StandardComparers/StringComparer.TcPOU
FUNCTION_BLOCK StringComparer EXTENDS Object IMPLEMENTS IComparer
VAR
	_ClassName : STRING := __POUNAME();
END_VAR

{attribute 'monitoring' := 'call'}
PROPERTY ClassName : STRING
GET
ClassName := _ClassName;
END_GET
END_PROPERTY

{attribute "object_name" := "Compare"}
METHOD Compare : COMPARISION_RESULT
VAR_INPUT
	left : PVOID;
	right : PVOID;
END_VAR
VAR
	leftPointer : POINTER TO STRING(255); 
	rightPointer : POINTER TO STRING(255); 
END_VAR
IF left = 0 AND right = 0 THEN
	Compare := COMPARISION_RESULT.EQUALS;
	RETURN;
END_IF

IF left = 0 THEN
	Compare := COMPARISION_RESULT.LEFT_LESS_RIGHT;
	RETURN;	
END_IF

IF right = 0 THEN
	Compare := COMPARISION_RESULT.LEFT_GREATER_RIGHT;
	RETURN;	
END_IF

leftPointer := left;
rightPointer := right;

IF leftPointer^ < rightPointer^ THEN
	Compare := COMPARISION_RESULT.LEFT_LESS_RIGHT;
ELSIF leftPointer^ > rightPointer^ THEN
	Compare := COMPARISION_RESULT.LEFT_GREATER_RIGHT;
ELSE
	Compare := COMPARISION_RESULT.EQUALS;	
END_IF
END_METHOD

END_FUNCTION_BLOCK

// ---- Comparing/StandardComparers/WStringComparer.TcPOU
FUNCTION_BLOCK WStringComparer EXTENDS Object IMPLEMENTS IComparer
VAR
	_ClassName : STRING := __POUNAME();
END_VAR

{attribute 'monitoring' := 'call'}
PROPERTY ClassName : STRING
GET
ClassName := _ClassName;
END_GET
END_PROPERTY

{attribute "object_name" := "Compare"}
METHOD Compare : COMPARISION_RESULT
VAR_INPUT
	left : PVOID;
	right : PVOID;
END_VAR
VAR
	leftPointer : POINTER TO WSTRING(255); 
	rightPointer : POINTER TO WSTRING(255); 
END_VAR
IF left = 0 AND right = 0 THEN
	Compare := COMPARISION_RESULT.EQUALS;
	RETURN;
END_IF

IF left = 0 THEN
	Compare := COMPARISION_RESULT.LEFT_LESS_RIGHT;
	RETURN;	
END_IF

IF right = 0 THEN
	Compare := COMPARISION_RESULT.LEFT_GREATER_RIGHT;
	RETURN;	
END_IF

leftPointer := left;
rightPointer := right;

IF leftPointer^ < rightPointer^ THEN
	Compare := COMPARISION_RESULT.LEFT_LESS_RIGHT;
ELSIF leftPointer^ > rightPointer^ THEN
	Compare := COMPARISION_RESULT.LEFT_GREATER_RIGHT;
ELSE
	Compare := COMPARISION_RESULT.EQUALS;	
END_IF
END_METHOD

END_FUNCTION_BLOCK

// ---- Comparing/StandardComparers/TimeComparer.TcPOU
FUNCTION_BLOCK TimeComparer EXTENDS Object IMPLEMENTS IComparer
VAR
	_ClassName : STRING := __POUNAME();
END_VAR

{attribute 'monitoring' := 'call'}
PROPERTY ClassName : STRING
GET
ClassName := _ClassName;
END_GET
END_PROPERTY

{attribute "object_name" := "Compare"}
METHOD Compare : COMPARISION_RESULT
VAR_INPUT
	left : PVOID;
	right : PVOID;
END_VAR
VAR
	leftPointer : POINTER TO TIME; 
	rightPointer : POINTER TO TIME; 
END_VAR
IF left = 0 AND right = 0 THEN
	Compare := COMPARISION_RESULT.EQUALS;
	RETURN;
END_IF

IF left = 0 THEN
	Compare := COMPARISION_RESULT.LEFT_LESS_RIGHT;
	RETURN;	
END_IF

IF right = 0 THEN
	Compare := COMPARISION_RESULT.LEFT_GREATER_RIGHT;
	RETURN;	
END_IF

leftPointer := left;
rightPointer := right;

IF leftPointer^ < rightPointer^ THEN
	Compare := COMPARISION_RESULT.LEFT_LESS_RIGHT;
ELSIF leftPointer^ > rightPointer^ THEN
	Compare := COMPARISION_RESULT.LEFT_GREATER_RIGHT;
ELSE
	Compare := COMPARISION_RESULT.EQUALS;	
END_IF
END_METHOD

END_FUNCTION_BLOCK

// ---- Comparing/StandardComparers/LTimeComparer.TcPOU
FUNCTION_BLOCK LTimeComparer EXTENDS Object IMPLEMENTS IComparer
VAR
	_ClassName : STRING := __POUNAME();
END_VAR

{attribute 'monitoring' := 'call'}
PROPERTY ClassName : STRING
GET
ClassName := _ClassName;
END_GET
END_PROPERTY

{attribute "object_name" := "Compare"}
METHOD Compare : COMPARISION_RESULT
VAR_INPUT
	left : PVOID;
	right : PVOID;
END_VAR
VAR
	leftPointer : POINTER TO LTIME; 
	rightPointer : POINTER TO LTIME; 
END_VAR
IF left = 0 AND right = 0 THEN
	Compare := COMPARISION_RESULT.EQUALS;
	RETURN;
END_IF

IF left = 0 THEN
	Compare := COMPARISION_RESULT.LEFT_LESS_RIGHT;
	RETURN;	
END_IF

IF right = 0 THEN
	Compare := COMPARISION_RESULT.LEFT_GREATER_RIGHT;
	RETURN;	
END_IF

leftPointer := left;
rightPointer := right;

IF leftPointer^ < rightPointer^ THEN
	Compare := COMPARISION_RESULT.LEFT_LESS_RIGHT;
ELSIF leftPointer^ > rightPointer^ THEN
	Compare := COMPARISION_RESULT.LEFT_GREATER_RIGHT;
ELSE
	Compare := COMPARISION_RESULT.EQUALS;	
END_IF
END_METHOD

END_FUNCTION_BLOCK

// ---- Comparing/StandardComparers/DateComparer.TcPOU
FUNCTION_BLOCK DateComparer EXTENDS Object IMPLEMENTS IComparer
VAR
	_ClassName : STRING := __POUNAME();
END_VAR

{attribute 'monitoring' := 'call'}
PROPERTY ClassName : STRING
GET
ClassName := _ClassName;
END_GET
END_PROPERTY

{attribute "object_name" := "Compare"}
METHOD Compare : COMPARISION_RESULT
VAR_INPUT
	left : PVOID;
	right : PVOID;
END_VAR
VAR
	leftPointer : POINTER TO DATE; 
	rightPointer : POINTER TO DATE; 
END_VAR
IF left = 0 AND right = 0 THEN
	Compare := COMPARISION_RESULT.EQUALS;
	RETURN;
END_IF

IF left = 0 THEN
	Compare := COMPARISION_RESULT.LEFT_LESS_RIGHT;
	RETURN;	
END_IF

IF right = 0 THEN
	Compare := COMPARISION_RESULT.LEFT_GREATER_RIGHT;
	RETURN;	
END_IF

leftPointer := left;
rightPointer := right;

IF leftPointer^ < rightPointer^ THEN
	Compare := COMPARISION_RESULT.LEFT_LESS_RIGHT;
ELSIF leftPointer^ > rightPointer^ THEN
	Compare := COMPARISION_RESULT.LEFT_GREATER_RIGHT;
ELSE
	Compare := COMPARISION_RESULT.EQUALS;	
END_IF
END_METHOD

END_FUNCTION_BLOCK

// ---- Comparing/StandardComparers/DateAndTimeComparer.TcPOU
FUNCTION_BLOCK DateAndTimeComparer EXTENDS Object IMPLEMENTS IComparer
VAR
	_ClassName : STRING := __POUNAME();
END_VAR

{attribute 'monitoring' := 'call'}
PROPERTY ClassName : STRING
GET
ClassName := _ClassName;
END_GET
END_PROPERTY

{attribute "object_name" := "Compare"}
METHOD Compare : COMPARISION_RESULT
VAR_INPUT
	left : PVOID;
	right : PVOID;
END_VAR
VAR
	leftPointer : POINTER TO DATE_AND_TIME; 
	rightPointer : POINTER TO DATE_AND_TIME; 
END_VAR
IF left = 0 AND right = 0 THEN
	Compare := COMPARISION_RESULT.EQUALS;
	RETURN;
END_IF

IF left = 0 THEN
	Compare := COMPARISION_RESULT.LEFT_LESS_RIGHT;
	RETURN;	
END_IF

IF right = 0 THEN
	Compare := COMPARISION_RESULT.LEFT_GREATER_RIGHT;
	RETURN;	
END_IF

leftPointer := left;
rightPointer := right;

IF leftPointer^ < rightPointer^ THEN
	Compare := COMPARISION_RESULT.LEFT_LESS_RIGHT;
ELSIF leftPointer^ > rightPointer^ THEN
	Compare := COMPARISION_RESULT.LEFT_GREATER_RIGHT;
ELSE
	Compare := COMPARISION_RESULT.EQUALS;	
END_IF
END_METHOD

END_FUNCTION_BLOCK

// ---- Comparing/StandardComparers/TimeOfDayComparer.TcPOU
FUNCTION_BLOCK TimeOfDayComparer EXTENDS Object IMPLEMENTS IComparer
VAR
	_ClassName : STRING := __POUNAME();
END_VAR

{attribute 'monitoring' := 'call'}
PROPERTY ClassName : STRING
GET
ClassName := _ClassName;
END_GET
END_PROPERTY

{attribute "object_name" := "Compare"}
METHOD Compare : COMPARISION_RESULT
VAR_INPUT
	left : PVOID;
	right : PVOID;
END_VAR
VAR
	leftPointer : POINTER TO TIME_OF_DAY; 
	rightPointer : POINTER TO TIME_OF_DAY; 
END_VAR
IF left = 0 AND right = 0 THEN
	Compare := COMPARISION_RESULT.EQUALS;
	RETURN;
END_IF

IF left = 0 THEN
	Compare := COMPARISION_RESULT.LEFT_LESS_RIGHT;
	RETURN;	
END_IF

IF right = 0 THEN
	Compare := COMPARISION_RESULT.LEFT_GREATER_RIGHT;
	RETURN;	
END_IF

leftPointer := left;
rightPointer := right;

IF leftPointer^ < rightPointer^ THEN
	Compare := COMPARISION_RESULT.LEFT_LESS_RIGHT;
ELSIF leftPointer^ > rightPointer^ THEN
	Compare := COMPARISION_RESULT.LEFT_GREATER_RIGHT;
ELSE
	Compare := COMPARISION_RESULT.EQUALS;	
END_IF
END_METHOD

END_FUNCTION_BLOCK

// ---- Comparing/StandardComparers/LTimeOfDayComparer.TcPOU
FUNCTION_BLOCK LTimeOfDayComparer EXTENDS Object IMPLEMENTS IComparer
VAR
	_ClassName : STRING := __POUNAME();
END_VAR

{attribute 'monitoring' := 'call'}
PROPERTY ClassName : STRING
GET
ClassName := _ClassName;
END_GET
END_PROPERTY

{attribute "object_name" := "Compare"}
METHOD Compare : COMPARISION_RESULT
VAR_INPUT
	left : PVOID;
	right : PVOID;
END_VAR
VAR
	leftPointer : POINTER TO LTIME_OF_DAY; 
	rightPointer : POINTER TO LTIME_OF_DAY; 
END_VAR
IF left = 0 AND right = 0 THEN
	Compare := COMPARISION_RESULT.EQUALS;
	RETURN;
END_IF

IF left = 0 THEN
	Compare := COMPARISION_RESULT.LEFT_LESS_RIGHT;
	RETURN;	
END_IF

IF right = 0 THEN
	Compare := COMPARISION_RESULT.LEFT_GREATER_RIGHT;
	RETURN;	
END_IF

leftPointer := left;
rightPointer := right;

IF leftPointer^ < rightPointer^ THEN
	Compare := COMPARISION_RESULT.LEFT_LESS_RIGHT;
ELSIF leftPointer^ > rightPointer^ THEN
	Compare := COMPARISION_RESULT.LEFT_GREATER_RIGHT;
ELSE
	Compare := COMPARISION_RESULT.EQUALS;	
END_IF
END_METHOD

END_FUNCTION_BLOCK

// ---- Comparing/StandardComparers/PointerComparer.TcPOU
FUNCTION_BLOCK PointerComparer EXTENDS Object IMPLEMENTS IComparer
VAR
	_ClassName : STRING := __POUNAME();
END_VAR

{attribute 'monitoring' := 'call'}
PROPERTY ClassName : STRING
GET
ClassName := _ClassName;
END_GET
END_PROPERTY

{attribute "object_name" := "Compare"}
METHOD Compare : COMPARISION_RESULT
VAR_INPUT
	left : PVOID;
	right : PVOID;
END_VAR
IF left < right THEN
	Compare := COMPARISION_RESULT.LEFT_LESS_RIGHT;
ELSIF left > right THEN
	Compare := COMPARISION_RESULT.LEFT_GREATER_RIGHT;
ELSE
	Compare := COMPARISION_RESULT.EQUALS;	
END_IF
END_METHOD

END_FUNCTION_BLOCK

// ---- Exceptions/Exception.TcPOU
{attribute 'enable_dynamic_creation'}	
{attribute 'no_explicit_call' := 'do not call this function block directly'} 
FUNCTION_BLOCK ABSTRACT Exception EXTENDS Object IMPLEMENTS IException
VAR
	_Fatal : BOOL; 	
	_SourceNamespaceName : STRING;
	_SourceClassName : STRING;
	_SourceMethodName : STRING;
	_SourcePosition : STRING;
	_LocalTimestamp : DATE_AND_TIME;	
	_UtcTimestamp : DATE_AND_TIME;	
END_VAR
VAR CONSTANT
	PATH_DELIMITER : WSTRING(1) := ".";
	UNSPECIFIED_METHOD : WSTRING(20) := "<unspecified method>";
	TIME_PREFIX : WSTRING(4) := " at ";
	SOURCE_PREFIX : WSTRING(4) := " in ";
	ERROR_CODE_PREFIX : WSTRING(13) := ", error code ";	
	LINE_NUMBER_PREFIX : WSTRING(13) := " line ";	
	INNER_MESSAGE_PREFIX : WSTRING(4) := " -> ";
END_VAR

METHOD PROTECTED AppendProgramOrganizationUnitFullName
VAR_IN_OUT CONSTANT
	stringBuilder : WideStringBuilder;
END_VAR
stringBuilder
	.AppendIf(_SourceNamespaceName, SourceNamespaceName <> '')
	.AppendStringIf(PATH_DELIMITER, SourceNamespaceName <> '')
	.AppendIf(_SourceClassName, SourceClassName <> '')
	.AppendStringIf(PATH_DELIMITER, SourceClassName <> '')
	.AppendIf(_SourceMethodName, SourceMethodName <> '')
	.AppendStringIf(UNSPECIFIED_METHOD, SourceMethodName = '');
END_METHOD

METHOD PROTECTED AppendSourceDescription
VAR_IN_OUT CONSTANT
	stringBuilder : WideStringBuilder;
END_VAR
AppendProgramOrganizationUnitFullName(stringBuilder);

stringBuilder
	.AppendStringIf(LINE_NUMBER_PREFIX, SourcePosition <> '')
	.AppendIf(_SourcePosition, SourcePosition <> '');
END_METHOD

METHOD PROTECTED AppendTimestampDescription
VAR_IN_OUT CONSTANT
	stringBuilder : WideStringBuilder;
END_VAR
stringBuilder
	.Append(_LocalTimestamp)
	.AppendString(" (")
	.Append(_UtcTimestamp)
	.AppendString("UTC)");
END_METHOD

METHOD ABSTRACT Clone : IObject
END_METHOD

{attribute 'monitoring' := 'call'}
PROPERTY ABSTRACT Empty : BOOL
GET
END_GET
END_PROPERTY

// Work is not possible after such error
{attribute 'monitoring' := 'call'}
PROPERTY Fatal : BOOL
GET
Fatal := _Fatal;
END_GET
SET // PROTECTED
_Fatal := Fatal;
END_SET
END_PROPERTY

METHOD ABSTRACT GetMessage : ERROR_MESSAGE
VAR_INPUT
	showTimestamp : BOOL := FALSE;
	showSource : BOOL := FALSE;
END_VAR
END_METHOD

METHOD GetSourceDescription : WSTRING(300)
VAR
	stringBuilder : WideStringBuilder;
END_VAR
AppendSourceDescription(stringBuilder);

stringBuilder.AssignToString(GetSourceDescription);
END_METHOD

{attribute 'monitoring' := 'call'}
PROPERTY LocalTimestamp : DATE_AND_TIME
GET
LocalTimestamp := _LocalTimestamp;
END_GET
SET // PROTECTED
_LocalTimestamp := LocalTimestamp;
END_SET
END_PROPERTY

{attribute 'monitoring' := 'call'}
PROPERTY SourceClassName : STRING
GET
SourceClassName := _SourceClassName;
END_GET
SET // PROTECTED
_SourceClassName := SourceClassName;
END_SET
END_PROPERTY

{attribute 'monitoring' := 'call'}
PROPERTY SourceMethodName : STRING
GET
SourceMethodName := _SourceMethodName;
END_GET
SET // PROTECTED
_SourceMethodName := SourceMethodName;
END_SET
END_PROPERTY

{attribute 'monitoring' := 'call'}
PROPERTY SourceNamespaceName : STRING
GET
SourceNamespaceName := _SourceNamespaceName;
END_GET
SET // PROTECTED
_SourceNamespaceName := SourceNamespaceName;
END_SET
END_PROPERTY

{attribute 'monitoring' := 'call'}
PROPERTY SourcePosition : STRING
GET
SourcePosition := _SourcePosition;
END_GET
SET // PROTECTED
_SourcePosition := SourcePosition;
END_SET
END_PROPERTY

{attribute 'monitoring' := 'call'}
PROPERTY UtcTimestamp : DATE_AND_TIME
GET
UtcTimestamp := _UtcTimestamp;
END_GET
SET // PROTECTED
_UtcTimestamp := UtcTimestamp;
END_SET
END_PROPERTY

END_FUNCTION_BLOCK

// ---- Primitives/String/StringBuilder.TcPOU
{attribute 'no_explicit_call' := 'Direct call is not allowed'} 
FUNCTION_BLOCK StringBuilder EXTENDS Object
VAR CONSTANT
	STRING_CHAR_SIZE : BYTE := 1;
END_VAR
VAR
	_ClassName : STRING := __POUNAME();

	_String : POINTER TO STRING;
	_Length : UDINT;
	_Capacity : UDINT;
END_VAR

METHOD Append : REFERENCE TO StringBuilder
VAR_INPUT
	value : ANY;
END_VAR
InternalAppend(value);

Append REF= THIS^;
END_METHOD

METHOD AppendIf : REFERENCE TO StringBuilder
VAR_INPUT
	value : ANY;
	condition : BOOL;
END_VAR
IF condition THEN
	InternalAppend(value);
END_IF

AppendIf REF= THIS^;
END_METHOD

METHOD AppendString : REFERENCE TO StringBuilder
VAR_IN_OUT CONSTANT
	value : STRING;
END_VAR
VAR
	valueDescriptor : __SYSTEM.AnyType;
END_VAR
valueDescriptor.TypeClass := __SYSTEM.TYPE_CLASS.TYPE_STRING;
valueDescriptor.pValue := ADR(value);
valueDescriptor.diSize := TO_DINT(Tc2_Utilities.LEN2(ADR(value))) + 1;

InternalAppend(valueDescriptor);

AppendString REF= THIS^;
END_METHOD

METHOD AppendStringIf : REFERENCE TO StringBuilder
VAR_IN_OUT CONSTANT
	value : STRING;
END_VAR
VAR_INPUT
	condition : BOOL;
END_VAR
VAR
	valueDescriptor : __SYSTEM.AnyType;
END_VAR
IF condition THEN
	valueDescriptor.TypeClass := __SYSTEM.TYPE_CLASS.TYPE_STRING;
	valueDescriptor.pValue := ADR(value);
	valueDescriptor.diSize := TO_DINT(Tc2_Utilities.LEN2(ADR(value))) + 1;
	
	InternalAppend(valueDescriptor);
END_IF

AppendStringIf REF= THIS^;
END_METHOD

METHOD AssignToString : BOOL
VAR_INPUT
	targetString : ANY_STRING;
END_VAR
VAR
	//exceptionFactory : ExceptionFactory(__POUNAME(), ClassName, CurrentNamespace.Name);
END_VAR
IF targetString.TypeClass <> __SYSTEM.TYPE_CLASS.TYPE_STRING THEN
	//exceptionFactory.ThrowException(__POSITION(), "Invalid string type, should be STRING");
END_IF

IF targetString.diSize < TO_DINT(_Length + STRING_CHAR_SIZE) THEN
	//exceptionFactory.ThrowException(__POSITION(), WStringHelper.Concat5("Target string size is ", TO_WSTRING(targetString.diSize), " bytes, but built string is ", TO_WSTRING(_Length + STRING_CHAR_SIZE), " bytes"));
END_IF

AssignToString := Tc2_Utilities.STRNCPY(targetString.pValue, _String, TO_UDINT(targetString.diSize));
END_METHOD

PROPERTY Capacity : UDINT
GET
Capacity := _Capacity;
END_GET
END_PROPERTY

{attribute 'monitoring' := 'call'}
PROPERTY ClassName : STRING
GET
ClassName := _ClassName;
END_GET
END_PROPERTY

METHOD Clear : REFERENCE TO StringBuilder
VAR_INPUT
	releaseMemory : BOOL;
END_VAR
_Length := 0;

IF _Capacity > 0 THEN
	IF releaseMemory THEN
		__DELETE(_String);	
		_Capacity := 0;	
	ELSE
		Tc2_System.MEMSET(_String, 0, StringMaxSize);
	END_IF	
END_IF

Clear REF= THIS^;
END_METHOD

METHOD ClearIf : REFERENCE TO StringBuilder
VAR_INPUT
	condition : BOOL;
	releaseMemory : BOOL;
END_VAR
IF condition THEN
	Clear(releaseMemory);
END_IF

ClearIf REF= THIS^;
END_METHOD

METHOD FB_exit : BOOL
VAR_INPUT
	bInCopyCode : BOOL; // if TRUE, the exit method is called for exiting an instance that is copied afterwards (online change).
END_VAR
Clear(TRUE);
END_METHOD

METHOD PROTECTED InternalAppend 
VAR_INPUT
	value : REFERENCE TO __System.AnyType;
END_VAR
VAR
	stringToAppend : STRING(255);	
	stringToAppendLength : UDINT;
	newString : POINTER TO BYTE;
	newCapacity : UDINT;
END_VAR
stringToAppend := StringHelper.InternalAnyToString(value);

stringToAppendLength := TO_UDINT(Tc2_Standard.LEN(stringToAppend));

IF _Capacity = 0 OR_ELSE _Length + stringToAppendLength > _Capacity THEN
	IF _Length + stringToAppendLength - _Capacity > 80 THEN
		newCapacity := _Length + stringToAppendLength;
	ELSE
		newCapacity := _Length + 80;
	END_IF
	
	newString := __NEW(BYTE, (STRING_CHAR_SIZE + (newCapacity * STRING_CHAR_SIZE)));
	
	IF _String <> 0 THEN
		Tc2_Utilities.STRNCPY(newString, _String, STRING_CHAR_SIZE + (newCapacity * STRING_CHAR_SIZE));
		
		__DELETE(_String);
	END_IF
	
	_String := newString;
	_Capacity := newCapacity;
END_IF

Tc2_Utilities.CONCAT2(_String, ADR(stringToAppend), _String, StringMaxSize);
_Length := _Length + stringToAppendLength;
END_METHOD

PROPERTY StringAddress : POINTER TO STRING
GET
StringAddress := _String;
END_GET
END_PROPERTY

PROPERTY StringLength : UDINT
GET
StringLength := _Length;
END_GET
END_PROPERTY

PROPERTY StringMaxSize : UDINT
GET
StringMaxSize := STRING_CHAR_SIZE + (STRING_CHAR_SIZE * _Capacity);
END_GET
END_PROPERTY

PROPERTY StringRealSize : UDINT
GET
StringRealSize := STRING_CHAR_SIZE + (STRING_CHAR_SIZE * _Length);
END_GET
END_PROPERTY

METHOD ToString255 : STRING(255)
IF _Length > 0 THEN
	Tc2_Utilities.STRNCPY(ADR(ToString255), _String, SIZEOF(ToString255));
END_IF
END_METHOD

END_FUNCTION_BLOCK

// ---- Primitives/String/StringHelper.TcPOU
{attribute 'no_explicit_call' := 'Direct call is not allowed'} 
PROGRAM StringHelper
VAR_OUTPUT
	NewLine : STRING(1) := F_ToChr(10);
END_VAR

METHOD AnyToString : STRING(255)
VAR_INPUT
	value : ANY;
END_VAR
AnyToString := InternalAnyToString(value);
END_METHOD

METHOD Append : BOOL
VAR_INPUT
	destinationString : ANY_STRING;
	sourceString : STRING(255);
END_VAR
VAR
	sources : ARRAY [1..1] OF POINTER TO STRING(255);
END_VAR
sources[1] := ADR(sourceString);

Append := InternalAppend(destinationString, sources);
END_METHOD

METHOD Append1 : BOOL
VAR_INPUT
	destinationString : ANY_STRING;
	sourceString1 : STRING(255);
END_VAR
VAR
	sources : ARRAY [1..1] OF POINTER TO STRING(255);
END_VAR
sources[1] := ADR(sourceString1);

Append1 := InternalAppend(destinationString, sources);
END_METHOD

METHOD Append10 : BOOL
VAR_INPUT
	destinationString : ANY_STRING;
	sourceString1 : STRING(255);
	sourceString2 : STRING(255);
	sourceString3 : STRING(255);
	sourceString4 : STRING(255);
	sourceString5 : STRING(255);
	sourceString6 : STRING(255);
	sourceString7 : STRING(255);
	sourceString8 : STRING(255);
	sourceString9 : STRING(255);
	sourceString10 : STRING(255);
END_VAR
VAR
	sources : ARRAY [1..10] OF POINTER TO STRING(255);
END_VAR
sources[1] := ADR(sourceString1);
sources[2] := ADR(sourceString2);
sources[3] := ADR(sourceString3);
sources[4] := ADR(sourceString4);
sources[5] := ADR(sourceString5);
sources[6] := ADR(sourceString6);
sources[7] := ADR(sourceString7);
sources[8] := ADR(sourceString8);
sources[9] := ADR(sourceString9);
sources[10] := ADR(sourceString10);

Append10 := InternalAppend(destinationString, sources);
END_METHOD

METHOD Append11 : BOOL
VAR_INPUT
	destinationString : ANY_STRING;
	sourceString1 : STRING(255);
	sourceString2 : STRING(255);
	sourceString3 : STRING(255);
	sourceString4 : STRING(255);
	sourceString5 : STRING(255);
	sourceString6 : STRING(255);
	sourceString7 : STRING(255);
	sourceString8 : STRING(255);
	sourceString9 : STRING(255);
	sourceString10 : STRING(255);
	sourceString11 : STRING(255);
END_VAR
VAR
	sources : ARRAY [1..11] OF POINTER TO STRING(255);
END_VAR
sources[1] := ADR(sourceString1);
sources[2] := ADR(sourceString2);
sources[3] := ADR(sourceString3);
sources[4] := ADR(sourceString4);
sources[5] := ADR(sourceString5);
sources[6] := ADR(sourceString6);
sources[7] := ADR(sourceString7);
sources[8] := ADR(sourceString8);
sources[9] := ADR(sourceString9);
sources[10] := ADR(sourceString10);
sources[11] := ADR(sourceString11);

Append11 := InternalAppend(destinationString, sources);
END_METHOD

METHOD Append12 : BOOL
VAR_INPUT
	destinationString : ANY_STRING;
	sourceString1 : STRING(255);
	sourceString2 : STRING(255);
	sourceString3 : STRING(255);
	sourceString4 : STRING(255);
	sourceString5 : STRING(255);
	sourceString6 : STRING(255);
	sourceString7 : STRING(255);
	sourceString8 : STRING(255);
	sourceString9 : STRING(255);
	sourceString10 : STRING(255);
	sourceString11 : STRING(255);
	sourceString12 : STRING(255);
END_VAR
VAR
	sources : ARRAY [1..12] OF POINTER TO STRING(255);
END_VAR
sources[1] := ADR(sourceString1);
sources[2] := ADR(sourceString2);
sources[3] := ADR(sourceString3);
sources[4] := ADR(sourceString4);
sources[5] := ADR(sourceString5);
sources[6] := ADR(sourceString6);
sources[7] := ADR(sourceString7);
sources[8] := ADR(sourceString8);
sources[9] := ADR(sourceString9);
sources[10] := ADR(sourceString10);
sources[11] := ADR(sourceString11);
sources[12] := ADR(sourceString12);

Append12 := InternalAppend(destinationString, sources);
END_METHOD

METHOD Append13 : BOOL
VAR_INPUT
	destinationString : ANY_STRING;
	sourceString1 : STRING(255);
	sourceString2 : STRING(255);
	sourceString3 : STRING(255);
	sourceString4 : STRING(255);
	sourceString5 : STRING(255);
	sourceString6 : STRING(255);
	sourceString7 : STRING(255);
	sourceString8 : STRING(255);
	sourceString9 : STRING(255);
	sourceString10 : STRING(255);
	sourceString11 : STRING(255);
	sourceString12 : STRING(255);
	sourceString13 : STRING(255);
END_VAR
VAR
	sources : ARRAY [1..13] OF POINTER TO STRING(255);
END_VAR
sources[1] := ADR(sourceString1);
sources[2] := ADR(sourceString2);
sources[3] := ADR(sourceString3);
sources[4] := ADR(sourceString4);
sources[5] := ADR(sourceString5);
sources[6] := ADR(sourceString6);
sources[7] := ADR(sourceString7);
sources[8] := ADR(sourceString8);
sources[9] := ADR(sourceString9);
sources[10] := ADR(sourceString10);
sources[11] := ADR(sourceString11);
sources[12] := ADR(sourceString12);
sources[13] := ADR(sourceString13);

Append13 := InternalAppend(destinationString, sources);
END_METHOD

METHOD Append14 : BOOL
VAR_INPUT
	destinationString : ANY_STRING;
	sourceString1 : STRING(255);
	sourceString2 : STRING(255);
	sourceString3 : STRING(255);
	sourceString4 : STRING(255);
	sourceString5 : STRING(255);
	sourceString6 : STRING(255);
	sourceString7 : STRING(255);
	sourceString8 : STRING(255);
	sourceString9 : STRING(255);
	sourceString10 : STRING(255);
	sourceString11 : STRING(255);
	sourceString12 : STRING(255);
	sourceString13 : STRING(255);
	sourceString14 : STRING(255);
END_VAR
VAR
	sources : ARRAY [1..14] OF POINTER TO STRING(255);
END_VAR
sources[1] := ADR(sourceString1);
sources[2] := ADR(sourceString2);
sources[3] := ADR(sourceString3);
sources[4] := ADR(sourceString4);
sources[5] := ADR(sourceString5);
sources[6] := ADR(sourceString6);
sources[7] := ADR(sourceString7);
sources[8] := ADR(sourceString8);
sources[9] := ADR(sourceString9);
sources[10] := ADR(sourceString10);
sources[11] := ADR(sourceString11);
sources[12] := ADR(sourceString12);
sources[13] := ADR(sourceString13);
sources[14] := ADR(sourceString14);

Append14 := InternalAppend(destinationString, sources);
END_METHOD

METHOD Append2 : BOOL
VAR_INPUT
	destinationString : ANY_STRING;
	sourceString1 : STRING(255);
	sourceString2 : STRING(255);
END_VAR
VAR
	sources : ARRAY [1..2] OF POINTER TO STRING(255);
END_VAR
sources[1] := ADR(sourceString1);
sources[2] := ADR(sourceString2);

Append2 := InternalAppend(destinationString, sources);
END_METHOD

METHOD Append3 : BOOL
VAR_INPUT
	destinationString : ANY_STRING;
	sourceString1 : STRING(255);
	sourceString2 : STRING(255);
	sourceString3 : STRING(255);
END_VAR
VAR
	sources : ARRAY [1..3] OF POINTER TO STRING(255);
END_VAR
sources[1] := ADR(sourceString1);
sources[2] := ADR(sourceString2);
sources[3] := ADR(sourceString3);

Append3 := InternalAppend(destinationString, sources);
END_METHOD

METHOD Append4 : BOOL
VAR_INPUT
	destinationString : ANY_STRING;
	sourceString1 : STRING(255);
	sourceString2 : STRING(255);
	sourceString3 : STRING(255);
	sourceString4 : STRING(255);
END_VAR
VAR
	sources : ARRAY [1..4] OF POINTER TO STRING(255);
END_VAR
sources[1] := ADR(sourceString1);
sources[2] := ADR(sourceString2);
sources[3] := ADR(sourceString3);
sources[4] := ADR(sourceString4);

Append4 := InternalAppend(destinationString, sources);
END_METHOD

METHOD Append5 : BOOL
VAR_INPUT
	destinationString : ANY_STRING;
	sourceString1 : STRING(255);
	sourceString2 : STRING(255);
	sourceString3 : STRING(255);
	sourceString4 : STRING(255);
	sourceString5 : STRING(255);
END_VAR
VAR
	sources : ARRAY [1..5] OF POINTER TO STRING(255);
END_VAR
sources[1] := ADR(sourceString1);
sources[2] := ADR(sourceString2);
sources[3] := ADR(sourceString3);
sources[4] := ADR(sourceString4);
sources[5] := ADR(sourceString5);

Append5 := InternalAppend(destinationString, sources);
END_METHOD

METHOD Append6 : BOOL
VAR_INPUT
	destinationString : ANY_STRING;
	sourceString1 : STRING(255);
	sourceString2 : STRING(255);
	sourceString3 : STRING(255);
	sourceString4 : STRING(255);
	sourceString5 : STRING(255);
	sourceString6 : STRING(255);
END_VAR
VAR
	sources : ARRAY [1..6] OF POINTER TO STRING(255);
END_VAR
sources[1] := ADR(sourceString1);
sources[2] := ADR(sourceString2);
sources[3] := ADR(sourceString3);
sources[4] := ADR(sourceString4);
sources[5] := ADR(sourceString5);
sources[6] := ADR(sourceString6);

Append6 := InternalAppend(destinationString, sources);
END_METHOD

METHOD Append7 : BOOL
VAR_INPUT
	destinationString : ANY_STRING;
	sourceString1 : STRING(255);
	sourceString2 : STRING(255);
	sourceString3 : STRING(255);
	sourceString4 : STRING(255);
	sourceString5 : STRING(255);
	sourceString6 : STRING(255);
	sourceString7 : STRING(255);
END_VAR
VAR
	sources : ARRAY [1..7] OF POINTER TO STRING(255);
END_VAR
sources[1] := ADR(sourceString1);
sources[2] := ADR(sourceString2);
sources[3] := ADR(sourceString3);
sources[4] := ADR(sourceString4);
sources[5] := ADR(sourceString5);
sources[6] := ADR(sourceString6);
sources[7] := ADR(sourceString7);

Append7 := InternalAppend(destinationString, sources);
END_METHOD

METHOD Append8 : BOOL
VAR_INPUT
	destinationString : ANY_STRING;
	sourceString1 : STRING(255);
	sourceString2 : STRING(255);
	sourceString3 : STRING(255);
	sourceString4 : STRING(255);
	sourceString5 : STRING(255);
	sourceString6 : STRING(255);
	sourceString7 : STRING(255);
	sourceString8 : STRING(255);
END_VAR
VAR
	sources : ARRAY [1..8] OF POINTER TO STRING(255);
END_VAR
sources[1] := ADR(sourceString1);
sources[2] := ADR(sourceString2);
sources[3] := ADR(sourceString3);
sources[4] := ADR(sourceString4);
sources[5] := ADR(sourceString5);
sources[6] := ADR(sourceString6);
sources[7] := ADR(sourceString7);
sources[8] := ADR(sourceString8);

Append8 := InternalAppend(destinationString, sources);
END_METHOD

METHOD Append9 : BOOL
VAR_INPUT
	destinationString : ANY_STRING;
	sourceString1 : STRING(255);
	sourceString2 : STRING(255);
	sourceString3 : STRING(255);
	sourceString4 : STRING(255);
	sourceString5 : STRING(255);
	sourceString6 : STRING(255);
	sourceString7 : STRING(255);
	sourceString8 : STRING(255);
	sourceString9 : STRING(255);
END_VAR
VAR
	sources : ARRAY [1..9] OF POINTER TO STRING(255);
END_VAR
sources[1] := ADR(sourceString1);
sources[2] := ADR(sourceString2);
sources[3] := ADR(sourceString3);
sources[4] := ADR(sourceString4);
sources[5] := ADR(sourceString5);
sources[6] := ADR(sourceString6);
sources[7] := ADR(sourceString7);
sources[8] := ADR(sourceString8);
sources[9] := ADR(sourceString9);

Append9 := InternalAppend(destinationString, sources);
END_METHOD

METHOD Concat10 : STRING(255)
VAR_INPUT
	string1 : STRING(255);
	string2 : STRING(255);
	string3 : STRING(255);
	string4 : STRING(255);
	string5 : STRING(255);
	string6 : STRING(255);
	string7 : STRING(255);
	string8 : STRING(255);
	string9 : STRING(255);
	string10 : STRING(255);
END_VAR
Concat10 := Tc2_Standard.CONCAT(
	Tc2_Standard.CONCAT(
		Tc2_Standard.CONCAT(Tc2_Standard.CONCAT(string1, string2), Tc2_Standard.CONCAT(string3, string4)), 
		Tc2_Standard.CONCAT(Tc2_Standard.CONCAT(string5, string6), Tc2_Standard.CONCAT(string7, string8)) 
	),
	Tc2_Standard.CONCAT(string9, string10));
END_METHOD

METHOD Concat11 : STRING(255)
VAR_INPUT
	string1 : STRING(255);
	string2 : STRING(255);
	string3 : STRING(255);
	string4 : STRING(255);
	string5 : STRING(255);
	string6 : STRING(255);
	string7 : STRING(255);
	string8 : STRING(255);
	string9 : STRING(255);
	string10 : STRING(255);
	string11 : STRING(255);
END_VAR
Concat11 := Tc2_Standard.CONCAT(
	Tc2_Standard.CONCAT(
		Tc2_Standard.CONCAT(Tc2_Standard.CONCAT(string1, string2), Tc2_Standard.CONCAT(string3, string4)), 
		Tc2_Standard.CONCAT(Tc2_Standard.CONCAT(string5, string6), Tc2_Standard.CONCAT(string7, string8)) 
	),
	Tc2_Standard.CONCAT(
		Tc2_Standard.CONCAT(string9, string10),
		string11
	)
);
END_METHOD

METHOD Concat12 : STRING(255)
VAR_INPUT
	string1 : STRING(255);
	string2 : STRING(255);
	string3 : STRING(255);
	string4 : STRING(255);
	string5 : STRING(255);
	string6 : STRING(255);
	string7 : STRING(255);
	string8 : STRING(255);
	string9 : STRING(255);
	string10 : STRING(255);
	string11 : STRING(255);
	string12 : STRING(255);
END_VAR
Concat12 := Tc2_Standard.CONCAT(
	Tc2_Standard.CONCAT(
		Tc2_Standard.CONCAT(Tc2_Standard.CONCAT(string1, string2), Tc2_Standard.CONCAT(string3, string4)), 
		Tc2_Standard.CONCAT(Tc2_Standard.CONCAT(string5, string6), Tc2_Standard.CONCAT(string7, string8)) 
	),
	Tc2_Standard.CONCAT(
		Tc2_Standard.CONCAT(string9, string10),
		Tc2_Standard.CONCAT(string11, string12)
	)
);
END_METHOD

METHOD Concat13 : STRING(255)
VAR_INPUT
	string1 : STRING(255);
	string2 : STRING(255);
	string3 : STRING(255);
	string4 : STRING(255);
	string5 : STRING(255);
	string6 : STRING(255);
	string7 : STRING(255);
	string8 : STRING(255);
	string9 : STRING(255);
	string10 : STRING(255);
	string11 : STRING(255);
	string12 : STRING(255);
	string13 : STRING(255);
END_VAR
Concat13 := Tc2_Standard.CONCAT(
	Tc2_Standard.CONCAT(
		Tc2_Standard.CONCAT(Tc2_Standard.CONCAT(string1, string2), Tc2_Standard.CONCAT(string3, string4)), 
		Tc2_Standard.CONCAT(Tc2_Standard.CONCAT(string5, string6), Tc2_Standard.CONCAT(string7, string8)) 
	),
	Tc2_Standard.CONCAT(
		Tc2_Standard.CONCAT(Tc2_Standard.CONCAT(string9, string10), Tc2_Standard.CONCAT(string11, string12)),
		string13
	)
);
END_METHOD

METHOD Concat14 : STRING(255)
VAR_INPUT
	string1 : STRING(255);
	string2 : STRING(255);
	string3 : STRING(255);
	string4 : STRING(255);
	string5 : STRING(255);
	string6 : STRING(255);
	string7 : STRING(255);
	string8 : STRING(255);
	string9 : STRING(255);
	string10 : STRING(255);
	string11 : STRING(255);
	string12 : STRING(255);
	string13 : STRING(255);
	string14 : STRING(255);
END_VAR
Concat14 := Tc2_Standard.CONCAT(
	Tc2_Standard.CONCAT(
		Tc2_Standard.CONCAT(Tc2_Standard.CONCAT(string1, string2), Tc2_Standard.CONCAT(string3, string4)), 
		Tc2_Standard.CONCAT(Tc2_Standard.CONCAT(string5, string6), Tc2_Standard.CONCAT(string7, string8)) 
	),
	Tc2_Standard.CONCAT(
		Tc2_Standard.CONCAT(Tc2_Standard.CONCAT(string9, string10), Tc2_Standard.CONCAT(string11, string12)),
		Tc2_Standard.CONCAT(string13, string14)
	)
);
END_METHOD

METHOD Concat2 : STRING(255)
VAR_INPUT
	string1 : STRING(255);
	string2 : STRING(255);
END_VAR
Concat2 := Tc2_Standard.CONCAT(string1, string2);
END_METHOD

METHOD Concat3 : STRING(255)
VAR_INPUT
	string1 : STRING(255);
	string2 : STRING(255);
	string3 : STRING(255);
END_VAR
Concat3 := Tc2_Standard.CONCAT(Tc2_Standard.CONCAT(string1, string2), string3);
END_METHOD

METHOD Concat4 : STRING(255)
VAR_INPUT
	string1 : STRING(255);
	string2 : STRING(255);
	string3 : STRING(255);
	string4 : STRING(255);
END_VAR
Concat4 := Tc2_Standard.CONCAT(Tc2_Standard.CONCAT(string1, string2), Tc2_Standard.CONCAT(string3, string4));
END_METHOD

METHOD Concat5 : STRING(255)
VAR_INPUT
	string1 : STRING(255);
	string2 : STRING(255);
	string3 : STRING(255);
	string4 : STRING(255);
	string5 : STRING(255);
END_VAR
Concat5 := Tc2_Standard.CONCAT(Tc2_Standard.CONCAT(Tc2_Standard.CONCAT(string1, string2), Tc2_Standard.CONCAT(string3, string4)), string5);
END_METHOD

METHOD Concat6 : STRING(255)
VAR_INPUT
	string1 : STRING(255);
	string2 : STRING(255);
	string3 : STRING(255);
	string4 : STRING(255);
	string5 : STRING(255);
	string6 : STRING(255);
END_VAR
Concat6 := Tc2_Standard.CONCAT(
	Tc2_Standard.CONCAT(Tc2_Standard.CONCAT(string1, string2), Tc2_Standard.CONCAT(string3, string4)), 
	Tc2_Standard.CONCAT(string5, string6)
);
END_METHOD

METHOD Concat7 : STRING(255)
VAR_INPUT
	string1 : STRING(255);
	string2 : STRING(255);
	string3 : STRING(255);
	string4 : STRING(255);
	string5 : STRING(255);
	string6 : STRING(255);
	string7 : STRING(255);
END_VAR
Concat7 := Tc2_Standard.CONCAT(
	Tc2_Standard.CONCAT(Tc2_Standard.CONCAT(string1, string2), Tc2_Standard.CONCAT(string3, string4)), 
	Tc2_Standard.CONCAT(Tc2_Standard.CONCAT(string5, string6), string7)
);
END_METHOD

METHOD Concat8 : STRING(255)
VAR_INPUT
	string1 : STRING(255);
	string2 : STRING(255);
	string3 : STRING(255);
	string4 : STRING(255);
	string5 : STRING(255);
	string6 : STRING(255);
	string7 : STRING(255);
	string8 : STRING(255);
END_VAR
Concat8 := Tc2_Standard.CONCAT(
	Tc2_Standard.CONCAT(Tc2_Standard.CONCAT(string1, string2), Tc2_Standard.CONCAT(string3, string4)), 
	Tc2_Standard.CONCAT(Tc2_Standard.CONCAT(string5, string6), Tc2_Standard.CONCAT(string7, string8)) 
);
END_METHOD

METHOD Concat9 : STRING(255)
VAR_INPUT
	string1 : STRING(255);
	string2 : STRING(255);
	string3 : STRING(255);
	string4 : STRING(255);
	string5 : STRING(255);
	string6 : STRING(255);
	string7 : STRING(255);
	string8 : STRING(255);
	string9 : STRING(255);
END_VAR
Concat9 := Tc2_Standard.CONCAT(
	Tc2_Standard.CONCAT(
		Tc2_Standard.CONCAT(Tc2_Standard.CONCAT(string1, string2), Tc2_Standard.CONCAT(string3, string4)), 
		Tc2_Standard.CONCAT(Tc2_Standard.CONCAT(string5, string6), Tc2_Standard.CONCAT(string7, string8)) 
	),
	string9);
END_METHOD

METHOD DateAndTimeToString : STRING
VAR_INPUT
	value : DATE_AND_TIME;
	dateValuesSeparator : STRING(1) := '_';
	dateAndTimeSeparator : STRING(1) := '-';
	timeValuesSeparator : STRING(1) := '_';
END_VAR
DateAndTimeToString := TO_STRING(value);

DateAndTimeToString := Tc2_Standard.DELETE(DateAndTimeToString, 3, 1);

DateAndTimeToString := Tc2_Standard.REPLACE(DateAndTimeToString, dateValuesSeparator, 1, 5);
DateAndTimeToString := Tc2_Standard.REPLACE(DateAndTimeToString, dateValuesSeparator, 1, 8);
DateAndTimeToString := Tc2_Standard.REPLACE(DateAndTimeToString, dateAndTimeSeparator, 1, 11);
DateAndTimeToString := Tc2_Standard.REPLACE(DateAndTimeToString, timeValuesSeparator, 1, 14);
DateAndTimeToString := Tc2_Standard.REPLACE(DateAndTimeToString, timeValuesSeparator, 1, 17);
END_METHOD

METHOD INTERNAL InternalAnyToString : STRING(255)
VAR_INPUT
	value : __System.AnyType;
END_VAR
VAR
	anyBool : POINTER TO BOOL;

	anyByte : POINTER TO BYTE;
	anyWord : POINTER TO WORD;
	anyDWord : POINTER TO LWORD;
	anyLWord : POINTER TO LWORD;
	
	anySInt : POINTER TO SINT;
	anyInt : POINTER TO INT;
	anyDInt : POINTER TO DINT;
	anyLInt : POINTER TO LINT;
	
	anyUSInt : POINTER TO USINT;
	anyUInt : POINTER TO UINT;
	anyUDInt : POINTER TO UDINT;
	anyULInt : POINTER TO ULINT;
	
	anyReal : POINTER TO REAL;
	anyLReal : POINTER TO LREAL;

	anyString : POINTER TO STRING(255);
	anyWString : POINTER TO WSTRING(255);
	
	anyTime : POINTER TO TIME;
	anyLTime : POINTER TO LTIME;
	anyDate : POINTER TO DATE;
	anyDateAndTime : POINTER TO DATE_AND_TIME;
	anyTimeOfDay : POINTER TO TOD;
END_VAR
CASE value.TypeClass OF
	__SYSTEM.TYPE_CLASS.TYPE_BOOL:
		anyBool := value.pValue;
		InternalAnyToString := TO_STRING(anyBool^);		
	
	__SYSTEM.TYPE_CLASS.TYPE_BIT:
		anyByte := value.pValue;
		IF anyByte^ > 0 THEN
			InternalAnyToString := '1';		
		ELSE
			InternalAnyToString := '0';		
		END_IF
	
	__SYSTEM.TYPE_CLASS.TYPE_BYTE:
		anyByte := value.pValue;
		InternalAnyToString := TO_STRING(anyByte^);		
	__SYSTEM.TYPE_CLASS.TYPE_WORD:
		anyWord := value.pValue;
		InternalAnyToString := TO_STRING(anyWord^);
	__SYSTEM.TYPE_CLASS.TYPE_DWORD:
		anyDWord := value.pValue;
		InternalAnyToString := TO_STRING(anyDWord^);
	__SYSTEM.TYPE_CLASS.TYPE_LWORD:
		anyLWord := value.pValue;
		InternalAnyToString := TO_STRING(anyLWord^);
		
	__SYSTEM.TYPE_CLASS.TYPE_SINT:
		anySInt := value.pValue;
		InternalAnyToString := TO_STRING(anySInt^);
	__SYSTEM.TYPE_CLASS.TYPE_INT:
		anyInt := value.pValue;
		InternalAnyToString := TO_STRING(anyInt^);		
	__SYSTEM.TYPE_CLASS.TYPE_DINT:
		anyDInt := value.pValue;
		InternalAnyToString := TO_STRING(anyDInt^);
	__SYSTEM.TYPE_CLASS.TYPE_LINT:
		anyLInt := value.pValue;
		InternalAnyToString := TO_STRING(anyLInt^);
		
	__SYSTEM.TYPE_CLASS.TYPE_USINT:
		anyUSInt := value.pValue;
		InternalAnyToString := TO_STRING(anyUSInt^);
	__SYSTEM.TYPE_CLASS.TYPE_UINT:
		anyUInt := value.pValue;
		InternalAnyToString := TO_STRING(anyUInt^);		
	__SYSTEM.TYPE_CLASS.TYPE_UDINT:
		anyUDInt := value.pValue;
		InternalAnyToString := TO_STRING(anyUDInt^);
	__SYSTEM.TYPE_CLASS.TYPE_ULINT:
		anyULInt := value.pValue;
		InternalAnyToString := TO_STRING(anyULInt^);

	__SYSTEM.TYPE_CLASS.TYPE_REAL:
		anyReal := value.pValue;
		InternalAnyToString := TO_STRING(anyReal^);
	__SYSTEM.TYPE_CLASS.TYPE_LREAL:
		anyLReal := value.pValue;
		InternalAnyToString := TO_STRING(anyLReal^);
	
	__SYSTEM.TYPE_CLASS.TYPE_STRING:
		anyString := value.pValue;
		InternalAnyToString := anyString^;
	__SYSTEM.TYPE_CLASS.TYPE_WSTRING:
		anyWString := value.pValue;
		InternalAnyToString := TO_STRING(anyWString^);
	
	__SYSTEM.TYPE_CLASS.TYPE_TIME:
		anyTime := value.pValue;
		InternalAnyToString := TO_STRING(anyTime^);
	__SYSTEM.TYPE_CLASS.TYPE_LTIME:
		anyLTime := value.pValue;
		InternalAnyToString := TO_STRING(anyLTime^);
	__SYSTEM.TYPE_CLASS.TYPE_DATE:
		anyDate := value.pValue;
		InternalAnyToString := TO_STRING(anyDate^);
	__SYSTEM.TYPE_CLASS.TYPE_DATEANDTIME:
		anyDateAndTime := value.pValue;
		InternalAnyToString := TO_STRING(anyDateAndTime^);  
	__SYSTEM.TYPE_CLASS.TYPE_TIMEOFDAY:
		anyTimeOfDay := value.pValue;
		InternalAnyToString := TO_STRING(anyTimeOfDay^);
	
	__SYSTEM.TYPE_CLASS.TYPE_POINTER, __SYSTEM.TYPE_CLASS.TYPE_REFERENCE:
		InternalAnyToString := Tc2_Utilities.PVOID_TO_HEXSTR(anyDate, 8, FALSE);		
	
	(*__SYSTEM.TYPE_CLASS.TYPE_SUBRANGE:
	__SYSTEM.TYPE_CLASS.TYPE_ENUM:
	__SYSTEM.TYPE_CLASS.TYPE_ARRAY:
	__SYSTEM.TYPE_CLASS.TYPE_PARAMS:
	__SYSTEM.TYPE_CLASS.TYPE_USERDEF:
	__SYSTEM.TYPE_CLASS.TYPE_NONE:
	__SYSTEM.TYPE_CLASS.TYPE_ANY:
	__SYSTEM.TYPE_CLASS.TYPE_ANYBIT:
	__SYSTEM.TYPE_CLASS.TYPE_ANYDATE:
	__SYSTEM.TYPE_CLASS.TYPE_ANYINT:
	__SYSTEM.TYPE_CLASS.TYPE_ANYNUM:
	__SYSTEM.TYPE_CLASS.TYPE_ANYREAL:
	__SYSTEM.TYPE_CLASS.TYPE_LAZY:
	__SYSTEM.TYPE_CLASS.TYPE_BITCONST:*)
	ELSE
		IF value.pValue <> 0 THEN
			InternalAnyToString := TO_STRING(value.pValue^); 
		ELSE
			InternalAnyToString := 'NULL';
		END_IF
END_CASE
END_METHOD

METHOD INTERNAL InternalAppend : BOOL
VAR_INPUT
	destinationString : __SYSTEM.AnyType;
END_VAR
VAR_IN_OUT
	sourceStrings : ARRAY [*] OF POINTER TO STRING(255);
END_VAR
VAR
	i : DINT;
END_VAR
IF destinationString.TypeClass <> __SYSTEM.TYPE_CLASS.TYPE_STRING THEN
	RETURN;
END_IF	

FOR i := LOWER_BOUND(sourceStrings, 1) TO UPPER_BOUND(sourceStrings, 1) DO
	InternalAppend := Tc2_Utilities.CONCAT2(destinationString.pValue, sourceStrings[i], destinationString.pValue, TO_UDINT(destinationString.diSize));	
END_FOR
END_METHOD

END_PROGRAM

// ---- Primitives/WideString/WideStringBuilder.TcPOU
{attribute 'no_explicit_call' := 'Direct call is not allowed'} 
FUNCTION_BLOCK WideStringBuilder EXTENDS Object
VAR CONSTANT
	STRING_CHAR_SIZE : BYTE := 2;
END_VAR
VAR
	_ClassName : STRING := __POUNAME();

	_String : POINTER TO WSTRING;
	_Length : UDINT;
	_Capacity : UDINT;
END_VAR

METHOD Append : REFERENCE TO WideStringBuilder
VAR_INPUT
	value : ANY;
END_VAR
InternalAppend(value);

Append REF= THIS^;
END_METHOD

METHOD AppendIf : REFERENCE TO WideStringBuilder
VAR_INPUT
	value : ANY;
	condition : BOOL;
END_VAR
IF condition THEN
	InternalAppend(value);
END_IF

AppendIf REF= THIS^;
END_METHOD

METHOD AppendString : REFERENCE TO WideStringBuilder
VAR_IN_OUT CONSTANT
	value : WSTRING;
END_VAR
VAR
	valueDescriptor : __SYSTEM.AnyType;
END_VAR
valueDescriptor.TypeClass := __SYSTEM.TYPE_CLASS.TYPE_WSTRING;
valueDescriptor.pValue := ADR(value);
valueDescriptor.diSize := 2 * TO_DINT(Tc2_Utilities.WLEN2(ADR(value))) + 2;

InternalAppend(valueDescriptor);

AppendString REF= THIS^;
END_METHOD

METHOD AppendStringIf : REFERENCE TO WideStringBuilder
VAR_IN_OUT CONSTANT
	value : WSTRING;
END_VAR
VAR_INPUT
	condition : BOOL;
END_VAR
VAR
	valueDescriptor : __SYSTEM.AnyType;
END_VAR
IF condition THEN
	valueDescriptor.TypeClass := __SYSTEM.TYPE_CLASS.TYPE_WSTRING;
	valueDescriptor.pValue := ADR(value);
	valueDescriptor.diSize := 2 * TO_DINT(Tc2_Utilities.WLEN2(ADR(value))) + 2;
	
	InternalAppend(valueDescriptor);
END_IF

AppendStringIf REF= THIS^;
END_METHOD

METHOD AssignToString : BOOL
VAR_INPUT
	targetString : ANY_STRING;
END_VAR
VAR
	//exceptionFactory : ExceptionFactory(__POUNAME(), ClassName, CurrentNamespace.Name);
END_VAR
IF targetString.TypeClass <> __SYSTEM.TYPE_CLASS.TYPE_WSTRING THEN
	//exceptionFactory.ThrowException(__POSITION(), "Invalid string type, should be WSTRING");
END_IF

IF targetString.diSize < TO_DINT(_Length + STRING_CHAR_SIZE) THEN
	//exceptionFactory.ThrowException(__POSITION(), WStringHelper.Concat5("Target string size is ", TO_WSTRING(targetString.diSize), " bytes, but built string is ", TO_WSTRING(_Length + STRING_CHAR_SIZE), " bytes"));
END_IF

AssignToString := Tc2_Utilities.WSTRNCPY(targetString.pValue, _String, TO_UDINT(targetString.diSize));
END_METHOD

PROPERTY Capacity : UDINT
GET
Capacity := _Capacity;
END_GET
END_PROPERTY

{attribute 'monitoring' := 'call'}
PROPERTY ClassName : STRING
GET
ClassName := _ClassName;
END_GET
END_PROPERTY

METHOD Clear : REFERENCE TO WideStringBuilder
VAR_INPUT
	releaseMemory : BOOL;
END_VAR
_Length := 0;

IF _Capacity > 0 THEN
	IF releaseMemory THEN
		__DELETE(_String);	
		_Capacity := 0;	
	ELSE
		Tc2_System.MEMSET(_String, 0, StringMaxSize);
	END_IF	
END_IF

Clear REF= THIS^;
END_METHOD

METHOD ClearIf : REFERENCE TO WideStringBuilder
VAR_INPUT
	condition : BOOL;
	releaseMemory : BOOL;
END_VAR
IF condition THEN
	Clear(releaseMemory);
END_IF

ClearIf REF= THIS^;
END_METHOD

METHOD FB_exit : BOOL
VAR_INPUT
	bInCopyCode : BOOL; // if TRUE, the exit method is called for exiting an instance that is copied afterwards (online change).
END_VAR
Clear(TRUE);
END_METHOD

METHOD PROTECTED InternalAppend 
VAR_INPUT
	value : REFERENCE TO __System.AnyType;
END_VAR
VAR
	stringToAppend : WSTRING(255);	
	stringToAppendLength : UDINT;
	newString : POINTER TO BYTE;
	newCapacity : UDINT;
END_VAR
stringToAppend := WideStringHelper.InternalAnyToString(value);

stringToAppendLength := TO_UDINT(Tc2_Standard.WLEN(stringToAppend));

IF _Capacity = 0 OR_ELSE _Length + stringToAppendLength > _Capacity THEN
	IF _Length + stringToAppendLength - _Capacity > 80 THEN
		newCapacity := _Length + stringToAppendLength;
	ELSE
		newCapacity := _Length + 80;
	END_IF
	
	newString := __NEW(BYTE, (STRING_CHAR_SIZE + (newCapacity * STRING_CHAR_SIZE)));
	
	IF _String <> 0 THEN
		Tc2_Utilities.WSTRNCPY(newString, _String, STRING_CHAR_SIZE + (newCapacity * STRING_CHAR_SIZE));
		
		__DELETE(_String);
	END_IF
	
	_String := newString;
	_Capacity := newCapacity;
END_IF

Tc2_Utilities.WCONCAT2(_String, ADR(stringToAppend), _String, StringMaxSize);
_Length := _Length + stringToAppendLength;
END_METHOD

PROPERTY StringAddress : POINTER TO WSTRING
GET
StringAddress := _String;
END_GET
END_PROPERTY

PROPERTY StringLength : UDINT
GET
StringLength := _Length;
END_GET
END_PROPERTY

PROPERTY StringMaxSize : UDINT
GET
StringMaxSize := STRING_CHAR_SIZE + (STRING_CHAR_SIZE * _Capacity);
END_GET
END_PROPERTY

PROPERTY StringRealSize : UDINT
GET
StringRealSize := STRING_CHAR_SIZE + (STRING_CHAR_SIZE * _Length);
END_GET
END_PROPERTY

METHOD ToString255 : WSTRING(255)
IF _Length > 0 THEN
	Tc2_Utilities.WSTRNCPY(ADR(ToString255), _String, SIZEOF(ToString255));
END_IF
END_METHOD

END_FUNCTION_BLOCK

// ---- Primitives/WideString/WideStringHelper.TcPOU
{attribute 'no_explicit_call' := 'Direct call is not allowed'} 
PROGRAM WideStringHelper
VAR_OUTPUT
	NewLine : WSTRING(1) := TO_WSTRING(Tc2_System.F_ToCHR(10)); 
END_VAR

METHOD AnyToString : WSTRING(255)
VAR_INPUT
	value : ANY;
END_VAR
AnyToString := InternalAnyToString(value);
END_METHOD

METHOD Append : BOOL
VAR_INPUT
	destinationString : ANY_STRING;
	sourceString : WSTRING(255);
END_VAR
VAR
	sources : ARRAY [1..1] OF POINTER TO WSTRING(255);
END_VAR
sources[1] := ADR(sourceString);

Append := InternalAppend(destinationString, sources);
END_METHOD

METHOD Append1 : BOOL
VAR_INPUT
	destinationString : ANY_STRING;
	sourceString1 : WSTRING(255);
END_VAR
VAR
	sources : ARRAY [1..1] OF POINTER TO WSTRING(255);
END_VAR
sources[1] := ADR(sourceString1);

Append1 := InternalAppend(destinationString, sources);
END_METHOD

METHOD Append10 : BOOL
VAR_INPUT
	destinationString : ANY_STRING;
	sourceString1 : WSTRING(255);
	sourceString2 : WSTRING(255);
	sourceString3 : WSTRING(255);
	sourceString4 : WSTRING(255);
	sourceString5 : WSTRING(255);
	sourceString6 : WSTRING(255);
	sourceString7 : WSTRING(255);
	sourceString8 : WSTRING(255);
	sourceString9 : WSTRING(255);
	sourceString10 : WSTRING(255);
END_VAR
VAR
	sources : ARRAY [1..10] OF POINTER TO WSTRING(255);
END_VAR
sources[1] := ADR(sourceString1);
sources[2] := ADR(sourceString2);
sources[3] := ADR(sourceString3);
sources[4] := ADR(sourceString4);
sources[5] := ADR(sourceString5);
sources[6] := ADR(sourceString6);
sources[7] := ADR(sourceString7);
sources[8] := ADR(sourceString8);
sources[9] := ADR(sourceString9);
sources[10] := ADR(sourceString10);

Append10 := InternalAppend(destinationString, sources);
END_METHOD

METHOD Append11 : BOOL
VAR_INPUT
	destinationString : ANY_STRING;
	sourceString1 : WSTRING(255);
	sourceString2 : WSTRING(255);
	sourceString3 : WSTRING(255);
	sourceString4 : WSTRING(255);
	sourceString5 : WSTRING(255);
	sourceString6 : WSTRING(255);
	sourceString7 : WSTRING(255);
	sourceString8 : WSTRING(255);
	sourceString9 : WSTRING(255);
	sourceString10 : WSTRING(255);
	sourceString11 : WSTRING(255);
END_VAR
VAR
	sources : ARRAY [1..11] OF POINTER TO WSTRING(255);
END_VAR
sources[1] := ADR(sourceString1);
sources[2] := ADR(sourceString2);
sources[3] := ADR(sourceString3);
sources[4] := ADR(sourceString4);
sources[5] := ADR(sourceString5);
sources[6] := ADR(sourceString6);
sources[7] := ADR(sourceString7);
sources[8] := ADR(sourceString8);
sources[9] := ADR(sourceString9);
sources[10] := ADR(sourceString10);
sources[11] := ADR(sourceString11);

Append11 := InternalAppend(destinationString, sources);
END_METHOD

METHOD Append12 : BOOL
VAR_INPUT
	destinationString : ANY_STRING;
	sourceString1 : WSTRING(255);
	sourceString2 : WSTRING(255);
	sourceString3 : WSTRING(255);
	sourceString4 : WSTRING(255);
	sourceString5 : WSTRING(255);
	sourceString6 : WSTRING(255);
	sourceString7 : WSTRING(255);
	sourceString8 : WSTRING(255);
	sourceString9 : WSTRING(255);
	sourceString10 : WSTRING(255);
	sourceString11 : WSTRING(255);
	sourceString12 : WSTRING(255);
END_VAR
VAR
	sources : ARRAY [1..12] OF POINTER TO WSTRING(255);
END_VAR
sources[1] := ADR(sourceString1);
sources[2] := ADR(sourceString2);
sources[3] := ADR(sourceString3);
sources[4] := ADR(sourceString4);
sources[5] := ADR(sourceString5);
sources[6] := ADR(sourceString6);
sources[7] := ADR(sourceString7);
sources[8] := ADR(sourceString8);
sources[9] := ADR(sourceString9);
sources[10] := ADR(sourceString10);
sources[11] := ADR(sourceString11);
sources[12] := ADR(sourceString12);

Append12 := InternalAppend(destinationString, sources);
END_METHOD

METHOD Append13 : BOOL
VAR_INPUT
	destinationString : ANY_STRING;
	sourceString1 : WSTRING(255);
	sourceString2 : WSTRING(255);
	sourceString3 : WSTRING(255);
	sourceString4 : WSTRING(255);
	sourceString5 : WSTRING(255);
	sourceString6 : WSTRING(255);
	sourceString7 : WSTRING(255);
	sourceString8 : WSTRING(255);
	sourceString9 : WSTRING(255);
	sourceString10 : WSTRING(255);
	sourceString11 : WSTRING(255);
	sourceString12 : WSTRING(255);
	sourceString13 : WSTRING(255);
END_VAR
VAR
	sources : ARRAY [1..13] OF POINTER TO WSTRING(255);
END_VAR
sources[1] := ADR(sourceString1);
sources[2] := ADR(sourceString2);
sources[3] := ADR(sourceString3);
sources[4] := ADR(sourceString4);
sources[5] := ADR(sourceString5);
sources[6] := ADR(sourceString6);
sources[7] := ADR(sourceString7);
sources[8] := ADR(sourceString8);
sources[9] := ADR(sourceString9);
sources[10] := ADR(sourceString10);
sources[11] := ADR(sourceString11);
sources[12] := ADR(sourceString12);
sources[13] := ADR(sourceString13);

Append13 := InternalAppend(destinationString, sources);
END_METHOD

METHOD Append14 : BOOL
VAR_INPUT
	destinationString : ANY_STRING;
	sourceString1 : WSTRING(255);
	sourceString2 : WSTRING(255);
	sourceString3 : WSTRING(255);
	sourceString4 : WSTRING(255);
	sourceString5 : WSTRING(255);
	sourceString6 : WSTRING(255);
	sourceString7 : WSTRING(255);
	sourceString8 : WSTRING(255);
	sourceString9 : WSTRING(255);
	sourceString10 : WSTRING(255);
	sourceString11 : WSTRING(255);
	sourceString12 : WSTRING(255);
	sourceString13 : WSTRING(255);
	sourceString14 : WSTRING(255);
END_VAR
VAR
	sources : ARRAY [1..14] OF POINTER TO WSTRING(255);
END_VAR
sources[1] := ADR(sourceString1);
sources[2] := ADR(sourceString2);
sources[3] := ADR(sourceString3);
sources[4] := ADR(sourceString4);
sources[5] := ADR(sourceString5);
sources[6] := ADR(sourceString6);
sources[7] := ADR(sourceString7);
sources[8] := ADR(sourceString8);
sources[9] := ADR(sourceString9);
sources[10] := ADR(sourceString10);
sources[11] := ADR(sourceString11);
sources[12] := ADR(sourceString12);
sources[13] := ADR(sourceString13);
sources[14] := ADR(sourceString14);

Append14 := InternalAppend(destinationString, sources);
END_METHOD

METHOD Append2 : BOOL
VAR_INPUT
	destinationString : ANY_STRING;
	sourceString1 : WSTRING(255);
	sourceString2 : WSTRING(255);
END_VAR
VAR
	sources : ARRAY [1..2] OF POINTER TO WSTRING(255);
END_VAR
sources[1] := ADR(sourceString1);
sources[2] := ADR(sourceString2);

Append2 := InternalAppend(destinationString, sources);
END_METHOD

METHOD Append3 : BOOL
VAR_INPUT
	destinationString : ANY_STRING;
	sourceString1 : WSTRING(255);
	sourceString2 : WSTRING(255);
	sourceString3 : WSTRING(255);
END_VAR
VAR
	sources : ARRAY [1..3] OF POINTER TO WSTRING(255);
END_VAR
sources[1] := ADR(sourceString1);
sources[2] := ADR(sourceString2);
sources[3] := ADR(sourceString3);

